// TwinCAT 3 PLC project WP_Controller
// ProgramVersion: 3.1.4024.0
// libraries:
//   CmpBitmapPool, * (System)
//   Tc2_EtherCAT, * (Beckhoff Automation GmbH)
//   Tc2_MC2, * (Beckhoff Automation GmbH)
//   Tc2_ModbusRTU, * (Beckhoff Automation GmbH)
//   Tc2_Standard, * (Beckhoff Automation GmbH)
//   Tc2_System, * (Beckhoff Automation GmbH)
//   Tc2_Utilities, * (Beckhoff Automation GmbH)
//   Tc3_Module, * (Beckhoff Automation GmbH)
//   Tc3_Vision, * (Beckhoff Automation GmbH)
// project tree:
//   DUTs/EtherCATDiagnostic/ E_EcDiacStatus.TcDUT (not stored), E_EcGetSlaveName.TcDUT (not stored), E_EcSystemStatus.TcDUT (not stored), ST_EcTerminalDiagInfo.TcDUT (not stored)
//   DUTs/TwinSAFE/ ST_AdsAddr.TcDUT (not stored)
//   DUTs/TwinSAFE/TwinSAFE_Connection/AX5805/ E_TsDiagnosisObjektsFA10AX5805.TcDUT, E_TsErrIndicesFA82AX5805.TcDUT, ST_TsConnectionInfoAX5805.TcDUT, ST_TsControlWordAX5805.TcDUT, ST_TsDiagObjectsFA10AX5805.TcDUT, ST_TsErrIndicesFA82AX5805.TcDUT, ST_TsSlaveInfoAX5805.TcDUT, ST_TsStatusWordAX5805.TcDUT
//   DUTs/TwinSAFE/TwinSAFE_Connection/EK1914/ ST_TsConnectionInfoEK1914.TcDUT, ST_TsDiagObjectsBitsEK1914.TcDUT, ST_TsDiagObjectsEK1914.TcDUT, ST_TsSlaveInfoEK1914.TcDUT
//   DUTs/TwinSAFE/TwinSAFE_Connection/EK1960/ ST_TsConnectionInfoEK1960.TcDUT, ST_TsDeviceInfoDataEK1960.TcDUT, ST_TsDiagObjectsEK1960.TcDUT, ST_TsSlaveInfoEK1960.TcDUT
//   DUTs/TwinSAFE/TwinSAFE_Connection/EL1904/ ST_TsConnectionInfoEL1904.TcDUT (not stored), ST_TsDiagObjectsBitsEL1904.TcDUT (not stored), ST_TsDiagObjectsEL1904.TcDUT (not stored), ST_TsSlaveInfoEL1904.TcDUT (not stored)
//   DUTs/TwinSAFE/TwinSAFE_Connection/EL1918/ ST_TsConnectionInfoEL1918.TcDUT, ST_TsDeviceInfoDataEL1918.TcDUT, ST_TsDiagObjectsEL1918.TcDUT, ST_TsSlaveInfoEL1918.TcDUT
//   DUTs/TwinSAFE/TwinSAFE_Connection/EL2904/ ST_TsConnectionInfoEL2904.TcDUT (not stored), ST_TsDiagObjectsBitsEL2904.TcDUT (not stored), ST_TsDiagObjectsEL2904.TcDUT (not stored), ST_TsSlaveInfoEL2904.TcDUT (not stored)
//   DUTs/TwinSAFE/TwinSAFE_Connection/EL2911/ ST_TsConnectionInfoEL2911.TcDUT, ST_TsDeviceInfoDataEL2911.TcDUT, ST_TsDiagObjectsEL2911.TcDUT, ST_TsSlaveInfoEL2911.TcDUT
//   DUTs/TwinSAFE/TwinSAFE_Connection/EL2912/ ST_TsConnectionInfoEL2912.TcDUT, ST_TsDeviceInfoDataEL2912.TcDUT, ST_TsDiagObjectsEL2912.TcDUT, ST_TsSlaveInfoEL2912.TcDUT
//   DUTs/TwinSAFE/TwinSAFE_Connection/EL3214/ ST_TsConnectionInfoEL3214.TcDUT, ST_TsSlaveInfoEL3214.TcDUT
//   DUTs/TwinSAFE/TwinSAFE_Connection/EL5021/ ST_TsConnectionInfoEL5021.TcDUT, ST_TsSlaveInfoEL5021.TcDUT
//   DUTs/TwinSAFE/TwinSAFE_Connection/EL6900/ ST_TsHardwareDiagC.TcDUT, ST_TsSlaveInfoEL6900.TcDUT
//   DUTs/TwinSAFE/TwinSAFE_Connection/EL6910/ ST_TsDeviceInfoDataC.TcDUT (not stored), ST_TsSlaveInfoEL6910.TcDUT (not stored)
//   DUTs/TwinSAFE/TwinSAFE_Connection/EP1957/ ST_TsConnectionInfoEP1957.TcDUT, ST_TsDeviceInfoDataEP1957.TcDUT, ST_TsDiagObjectsEP1957.TcDUT, ST_TsSlaveInfoEP1957.TcDUT
//   DUTs/TwinSAFE/TwinSAFE_Connection/ E_TsCycleDiagObj.TcDUT (not stored), ST_TsConnectionInfo12Byte.TcDUT (not stored), ST_TsConnectionInfo1Byte.TcDUT (not stored), ST_TsConnectionInfo2Byte.TcDUT (not stored), ST_TsConnectionInfo4Byte.TcDUT (not stored), ST_TsConnectionInfo8Byte.TcDUT (not stored), ST_TsSlave2Temp.TcDUT (not stored), ST_TsSlave3Temp.TcDUT (not stored), ST_TsSlaveAddress.TcDUT (not stored), ST_TsSlaveAddressCRC.TcDUT (not stored)
//   DUTs/TwinSAFE/TwinSAFE_Functionblocks/ E_TsFbType.TcDUT (not stored), ST_TsFbInfo.TcDUT (not stored)
//   DUTs/TwinSAFE/TwinSAFE_Group/ ST_TsGroupInfo.TcDUT (not stored)
//   GVLs/ GVL.TcGVL, IO.TcGVL
//   / PlcTask.TcTTO (not stored), VisionTask.TcTTO (not stored)
//   POUs/ FB_ClockPulse.TcPOU, FB_EnableAxes.TcPOU (not stored), FB_StrASCConversion.TcPOU (not stored), F_Scale.TcPOU (not stored), MAIN.TcPOU, PRG_LoadcellScaling.TcPOU, PRG_MotorDrive.TcPOU, PRG_PLCModbusRTU.TcPOU, PRG_PneumaticValves.TcPOU, PRG_PowerMeasurement.TcPOU, PRG_SafetyLightCurtain.TcPOU, PRG_Thermocouple.TcPOU, PRG_VfdModbusRtu.TcPOU, VISION.TcPOU, Vision_test.TcPOU
//   POUs/TwinSAFE/ FB_EcGetSlaveName.TcPOU, FB_TwinSafeConnectionEL1904.TcPOU (not stored), FB_TwinSafeConnectionEL2912.TcPOU, FB_TwinSafeConnectionEL6910.TcPOU (not stored), FB_TwinSafeFB.TcPOU (not stored), FB_TwinSafeGroup.TcPOU (not stored), FB_TwinSafeGroupExt.TcPOU (not stored)
// real-time tasks:
//   TASK PlcTask: cycle T#10ms, priority 20, ADS port 350
//   TASK VisionTask: cycle T#10ms, priority 21, ADS port 351
//   TASK VnTask ImgAcq (Camera1): cycle T#1ms, priority 5, ADS port 352
//   TASK VnTask ADS (Camera1): cycle T#10ms, priority 6, ADS port 353
//   TASK VnTask ImgAcq (FileSource1): cycle T#10ms, priority 7, ADS port 354
// motion (NC):
//   TASK NC-Task 1 SAF: cycle T#2ms, priority 4, ADS port 501
//   TASK NC-Task 1 SVB: cycle T#10ms, priority 8, ADS port 511
//   AXIS Axis 1 (id 1)
//     General: UnitName=°
//     Dynamic: AccelerationMaximum=52000, DecelerationMaximum=52000, Acceleration=49770, Deceleration=49770, Jerk=149310
//     Velo: RefSearch=331.8, RefSync=331.8, SlowManual=1659, FastManual=9954, Fast=33180, Maximum=33180
//     OtherSettings: AllowMotionCmdToSlave=true
//     encoder EncType=19
//       EncPara: ScaleFactorNumerator=360, ScaleFactorDenominator=1048576, MaxCount=#xffffffff
//         TimeComp: TimeCompMode=1, EncDelayCycles=4
//     drive DrvType=16
//       DrvPara: MaxCount=#xffffffff, DriveControlDWord=#x00020000
//         Analog: VeloReferenz=36498, VeloScale=32, TorqueSetpointScale=10, ScaleFactorActTorque=0.1
//         TimeComp: TaskDelayCycles=1
//     controller CtrType=1
//       CtrPara: PriorControlFactor=1
//         PosDiffControl: Enable=false
//         Observer: BandWidth=20
// I/O:
//   DEVICE Device 5 (EtherCAT), AmsNetId 169.254.69.6.6.1
//     Term 12 (EK1100) [EK1100 EtherCAT Coupler (2A E-Bus)]
//       Term 13 (EL1809) [EL1809 16Ch. Dig. Input 24V, 3ms]
//       Term 14 (EL2809-0015) [EL2809-0015 16Ch. Dig. Output 24V DC, 0.35A, not short-circuit proof]
//       Term 15 (EL6910) [EL6910, TwinSAFE PLC]
//       Term 16 (EL1904) [EL1904, 4 Ch. Safety Input 24V, TwinSAFE]
//         modules: Module 1 (FSOES)
//       Term 17 (EL2912) [EL2912, 2Ch. Safety Output 24V, 2A, TwinSAFE]
//         modules: Module 1 (FSOE), Module 2 (FSOUT), Module 3 (DEVICEIO), Module 4 (FSLOGIC)
//       Term 18 (EL3443) [EL3443 3Ch. Power Measuring]
//       Term 19 (EL3312) [EL3312 2Ch. Ana. Input Thermocouple (TC)]
//       Term 20 (EL6021) [EL6021 Interface (RS422/485)]
//       Term 21 (EL6021) [EL6021 Interface (RS422/485)]
//       Term 22 (EL9410) [EL9410 E-Bus Power Supplier  (Diagnostics)]
//       Term 23 (EL7221-9014) [EL7221-9014 1Ch. MDP742 Servo motor output stage with OCT (50V, 8A RMS) and STO input]
//       Term 24 (EL7221-9014) [EL7221-9014 1Ch. MDP742 Servo motor output stage with OCT (50V, 8A RMS) and STO input]
//       Term 25 (EL9512) [EL9512 Power supply terminal 12V]
//       Term 26 (EL3356-0010) [EL3356-0010 1Ch. Ana. Input Resistor Bridge Terminal, 24bit, High Precision]
//       Term 27 (EL9011) [EL9011 End Terminal]
// variable links:
//   NC-Task 1 SAF/Axes/Axis 1 <-> Device 5 (EtherCAT)/Term 12 (EK1100)/Term 23 (EL7221-9014)
//     Drive/Inputs/In/nDcOutputTime <-> InfoData/DcOutputShift
//     Drive/Inputs/In/nState1 <-> DRV Statusword/Statusword
//     Drive/Inputs/In/nState2 <-> DRV Statusword/Statusword @bit 8
//     Drive/Inputs/In/nState4 @bit 1 <-> WcState/InputToggle
//     Drive/Inputs/In/nState4 <-> WcState/WcState
//     Drive/Outputs/Out/nCtrl1 <-> DRV Controlword/Controlword
//     Drive/Outputs/Out/nCtrl2 <-> DRV Controlword/Controlword @bit 8
//     Drive/Outputs/Out/nDataOut2 <-> DRV Target velocity/Target velocity
//     Enc/Inputs/In/nDataIn1 <-> FB Position/Position
//     Enc/Inputs/In/nDcInputTime <-> InfoData/DcInputShift
//     Enc/Inputs/In/nState4 @bit 1 <-> WcState/InputToggle
//     Enc/Inputs/In/nState4 <-> WcState/WcState
//   WP_Controller/WP_Controller Instance <-> Device 5 (EtherCAT)/Term 12 (EK1100)/Term 14 (EL2809-0015)
//     PlcTask Outputs/GVL.bFan <-> Channel 9/Output
//     PlcTask Outputs/GVL.bLight <-> Channel 8/Output
//   WP_Controller/WP_Controller Instance <-> Device 5 (EtherCAT)/Term 12 (EK1100)/Term 18 (EL3443)
//     PlcTask Inputs/GVL.fActivePower <-> L1 Power/Active Power
//     PlcTask Inputs/GVL.fIL1 <-> L1 Basic/Current
//     VisionTask Inputs/GVL.fFrequency <-> Total Basic/Frequency
//     VisionTask Inputs/GVL.fUL1 <-> L1 Basic/Voltage
//     VisionTask Inputs/GVL.fcosphi1 <-> L1 Power/Power Factor
//   WP_Controller/WP_Controller Instance <-> Device 5 (EtherCAT)/Term 12 (EK1100)/Term 19 (EL3312)
//     PlcTask Inputs/GVL.nTemp <-> TC Inputs Channel 1/Value
//   WP_Controller/WP_Controller Instance <-> Device 5 (EtherCAT)/Term 12 (EK1100)/Term 20 (EL6021)
//     PlcTask Inputs/PRG_VfdModbusRtu.fbVfdMb.InData/D <-> COM TxPDO-Map Inputs/Data In 0
//     PlcTask Inputs/PRG_VfdModbusRtu.fbVfdMb.InData/D @bit {8..168 step 8} <-> COM TxPDO-Map Inputs/Data In {1..21}  (21 links)
//     PlcTask Inputs/PRG_VfdModbusRtu.fbVfdMb.InData/Status <-> COM TxPDO-Map Inputs/Status
//     PlcTask Outputs/PRG_VfdModbusRtu.fbVfdMb.OutData/Ctrl <-> COM RxPDO-Map Outputs/Ctrl
//     PlcTask Outputs/PRG_VfdModbusRtu.fbVfdMb.OutData/D <-> COM RxPDO-Map Outputs/Data Out 0
//     PlcTask Outputs/PRG_VfdModbusRtu.fbVfdMb.OutData/D @bit {8..168 step 8} <-> COM RxPDO-Map Outputs/Data Out {1..21}  (21 links)
//   WP_Controller/WP_Controller Instance <-> Device 5 (EtherCAT)/Term 12 (EK1100)/Term 21 (EL6021)
//     PlcTask Inputs/PRG_PLCModbusRTU.fbModbusMaster.InData/D <-> COM TxPDO-Map Inputs/Data In 0
//     PlcTask Inputs/PRG_PLCModbusRTU.fbModbusMaster.InData/D @bit {8..168 step 8} <-> COM TxPDO-Map Inputs/Data In {1..21}  (21 links)
//     PlcTask Inputs/PRG_PLCModbusRTU.fbModbusMaster.InData/Status <-> COM TxPDO-Map Inputs/Status
//     PlcTask Outputs/PRG_PLCModbusRTU.fbModbusMaster.OutData/Ctrl <-> COM RxPDO-Map Outputs/Ctrl
//     PlcTask Outputs/PRG_PLCModbusRTU.fbModbusMaster.OutData/D <-> COM RxPDO-Map Outputs/Data Out 0
//     PlcTask Outputs/PRG_PLCModbusRTU.fbModbusMaster.OutData/D @bit {8..168 step 8} <-> COM RxPDO-Map Outputs/Data Out {1..21}  (21 links)
//   WP_Controller/WP_Controller Instance <-> Device 5 (EtherCAT)/Term 12 (EK1100)/Term 26 (EL3356-0010)
//     PlcTask Inputs/GVL.uLoadCellRawValue <-> RMB Value (INT32)/Value
//   WP_Controller/WP_Controller Instance <-> NC-Task 1 SAF/Axes/Axis 1
//     PlcTask Inputs/GVL.stAxis1.NcToPlc <-> Outputs/ToPlc
//     PlcTask Outputs/GVL.stAxis1.PlcToNc <-> Inputs/FromPlc

// ---- DUTs/TwinSAFE/TwinSAFE_Connection/AX5805/E_TsDiagnosisObjektsFA10AX5805.TcDUT
TYPE E_TsDiagnosisObjektsFA10AX5805 :
(*******************************************************************************************************
Description			:	Reason for shutdown of CoE objects 0xFA10
Supported terminals : 	AX5805, AX5806
Documentation 		:	AX5805 / AX5806 TwinSAFE drive option cards for the AX5000 servo drive
Version/Date 		:	V1.6.1/15.03.2016
********************************************************************************************************)
(

	eFA10AX5805_NoErrorReaction					:= 16#0000,	(* Error reaction: no error reaction *)
	eFA10AX5805_ErrSafeTorqueOff				:= 16#0040,	(* Error reaction: STO (Safe Torque Off) *)
	eFA10AX5805_ErrSafeStop1					:= 16#0050,	(* Error reaction: SS1 (Safe Stop 1) *)

	eFA10AX5805_StatusWordIncorrect				:= 16#0100,	(* Shutdown reason: The status word was calculated incorrectly *)
	eFA10AX5805_ParametersWrongOrNotLoaded		:= 16#0200,	(* Shutdown reason: The parameters are wrong or not yet loaded *)
	eFA10AX5805_FSOEProtocolWrongState			:= 16#0300,	(* Shutdown reason: FSOE protocol not in state DATA *)
	eFA10AX5805_WrongDriveParameter				:= 16#0400,	(* Shutdown reason: Internal comparison failed. Please check the motor/drive dimensioning/parameterization *)
	eFA10AX5805_ExtCamDetectedUnexpectedly		:= 16#0500,	(* Reason for shutdown position detection: external cam detected unexpectedly *)
	eFA10AX5805_ExtCamRightSideCamWindow		:= 16#0600,	(* Reason for shutdown position detection: external cam detected to the right of the cam window *)
	eFA10AX5805_ExtCamLeftSideCamWindow			:= 16#0700,	(* Reason for shutdown position detection: external cam detected to the left of the cam window *)
	eFA10AX5805_MaxTraversingRangeExceeded		:= 16#0800,	(* Reason for shutdown position detection: the maximum traversing range was exceeded *)
	eFA10AX5805_SS1SwitchedOff					:= 16#5000,	(* Reason for shutdown safety function: The safety function SS1 has switched off *)
	eFA10AX5805_SOSSwitchedOff					:= 16#6800,	(* Reason for shutdown safety function: The safety function SOS has switched off *)
	eFA10AX5805_SSRSwitchedOff					:= 16#8000,	(* Reason for shutdown safety function: The safety function SSR has switched off *)
	eFA10AX5805_SLSSwitchedOff					:= 16#9000,	(* Reason for shutdown safety function: The safety function SLS has switched off *)
	eFA10AX5805_SLPSwitchedOff					:= 16#A000,	(* Reason for shutdown safety function: The safety function SLP has switched off *)
	eFA10AX5805_SMSSwitchedOff					:= 16#A800,	(* Reason for shutdown safety function: The safety function SMS has switched off *)
	eFA10AX5805_SLISwitchedOff					:= 16#B800,	(* Reason for shutdown safety function: The safety function SLI has switched off *)
	eFA10AX5805_SARSwitchedOff					:= 16#C000,	(* Reason for shutdown safety function: The safety function SAR has switched off *)
	eFA10AX5805_SMASwitchedOff					:= 16#C800,	(* Reason for shutdown safety function: The safety function SMA has switched off *)
	eFA10AX5805_SDIpSwitchedOff					:= 16#D000,	(* Reason for shutdown safety function: The safety function SDIp has switched off *)
	eFA10AX5805_SDInSwitchedOff					:= 16#D100	(* Reason for shutdown safety function: The safety function SDIn has switched off *)
	
);
END_TYPE
(* End *)

// ---- DUTs/TwinSAFE/TwinSAFE_Connection/AX5805/E_TsErrIndicesFA82AX5805.TcDUT
TYPE E_TsErrIndicesFA82AX5805 :
(*******************************************************************************************************
Description			:	Error indices in CoE objects 0xFA82
Supported terminals : 	AX5805, AX5806
Documentation 		:	AX5805 / AX5806 TwinSAFE drive option cards for the AX5000 servo drive
Version/Date 		:	V1.6.1/15.03.2016
********************************************************************************************************)
(

	eAX5805FA82_NoError									:=	16#0000,	

	eAX5805FA82_FAULT_MAXT_C1							:=	16#0001,	(* The temperature has exceeded the maximum permissible temperature (µC1) *)
	eAX5805FA82_FAULT_MAXT_C2							:=	16#0002,	(* The temperature has exceeded the maximum permissible temperature (µC2) *)
	eAX5805FA82_FAULT_MINT_C1							:=	16#0003,	(* The temperature has fallen below the minimum permissible temperature (µC1) *)
	eAX5805FA82_FAULT_MINT_C2							:=	16#0004,	(* The temperature has fallen below the minimum permissible temperature (µC2) *)

	eAX5805FA82_HW_ERR_MAX_VCC_C1						:=	16#0101,	(* The maximum supply voltage was exceeded (3.3 V) *)
	eAX5805FA82_HW_ERR_MAX_VCC_C2						:=	16#0102,	(* The maximum supply voltage was exceeded (3.3 V) *)
	eAX5805FA82_HW_ERR_MIN_VCC_C1						:=	16#0103,	(* The supply voltage fell below the minimum value (3.3 V) *)
	eAX5805FA82_HW_ERR_MIN_VCC_C2						:=	16#0104,	(* The supply voltage fell below the minimum value (3.3 V) *)

	eAX5805FA82_FAULT_MCTC1_TO							:=	16#0201,	(* The MCTests of µC1 were not carried out completely within the specified time *)
	eAX5805FA82_FAULT_MCTC2_TO							:=	16#0202,	(* The MCTests of µC2 were not carried out completely within the specified time *)
	eAX5805FA82_FAULT_TIMER_C1							:=	16#0203,	(* The global timer was not updated in time *)
	eAX5805FA82_FAULT_TIMER_C2							:=	16#0204,	(* The global timer was not updated in time *)
	eAX5805FA82_FAULT_TS_WDG_TO_C1						:=	16#020C,	(* The TwinSAFE module was not called within the watchdog time *)
	eAX5805FA82_FAULT_TS_WDG_TO_C2						:=	16#020D,	(* The TwinSAFE module was not called within the watchdog time *)
	eAX5805FA82_FAULT_RESET_MC1							:=	16#020E,	(* A reset has occurred in the operation of the controller for µC1. µC2 was not reset thereby *)
	
	eAX5805FA82_FAULT_SERCOMC2							:=	16#0300,	(* An error occurred in the SerComP24C2 module during data transmission *)

	eAX5805FA82_FAULT_SERCOM_1							:=	16#0401,	(* An error occurred in the SerComP24C1 module during data transmission *)
	eAX5805FA82_FAULT_SERCOM_2							:=	16#0402,	(* An error occurred in the SerComP24C1 module during data transmission *)
	eAX5805FA82_FAULT_SERCOM_3							:=	16#0403,	(* An error occurred in the SerComP24C1 module during data transmission *)
	eAX5805FA82_FAULT_SERCOM_4							:=	16#0404,	(* An error occurred in the SerComP24C1 module during data transmission *)
	eAX5805FA82_FAULT_SERCOM_5							:=	16#0405,	(* An error occurred in the SerComP24C1 module during data transmission *)
	eAX5805FA82_FAULT_SERCOM_6							:=	16#0406,	(* An error occurred in the SerComP24C1 module during data transmission *)
	eAX5805FA82_FAULT_SERCOM_7							:=	16#0407,	(* An error occurred in the SerComP24C1 module during data transmission *)
	eAX5805FA82_FAULT_SERCOM_8							:=	16#0408,	(* An error occurred in the SerComP24C1 module during data transmission *)
	eAX5805FA82_FAULT_SERCOM_9							:=	16#0409,	(* An error occurred in the SerComP24C1 module during data transmission *)
	eAX5805FA82_FAULT_SERCOM_A							:=	16#040A,	(* An error occurred in the SerComP24C1 module during data transmission *)
	eAX5805FA82_FAULT_SERCOM_B							:=	16#040B,	(* An error occurred in the SerComP24C1 module during data transmission *)

	eAX5805FA82_FAULT_TEMPSENSOR_1						:=	16#0501,	(* Error in the communication with one of the temperature sensors *)
	eAX5805FA82_FAULT_TEMPSENSOR_2						:=	16#0502,	(* Error in the communication with one of the temperature sensors *)
	eAX5805FA82_FAULT_TEMPSENSOR_3						:=	16#0503,	(* Error in the communication with one of the temperature sensors *)
	eAX5805FA82_FAULT_TEMPSENSOR_4						:=	16#0504,	(* Error in the communication with one of the temperature sensors *)
	eAX5805FA82_FAULT_TEMPSENSOR_5						:=	16#0505,	(* Error in the communication with one of the temperature sensors *)
	eAX5805FA82_FAULT_TEMPSENSOR_6						:=	16#0506,	(* Error in the communication with one of the temperature sensors *)
	eAX5805FA82_FAULT_TEMPSENSOR_7						:=	16#0507,	(* Error in the communication with one of the temperature sensors *)

	eAX5805FA82_FAULT_OUTPUTCOMPARE						:=	16#0601,	(* The values output by µC1 and µC2 differ *)
	eAX5805FA82_FAULT_OUTPUTCOMPAREC2					:=	16#0602,	(* The values output by µC1 and µC2 differ *)

	eAX5805FA82_HW_ERR_MIN_VCC_FPGA						:=	16#0700,	(* The FPGA supply voltage fell below the minimum value (5 V) *)
	eAX5805FA82_HW_ERR_MAX_VCC_FPGA						:=	16#0701,	(* The FPGA supply voltage exceeded the maximum value (5 V) *)

	eAX5805FA82_FAULT_FEEDBACK_C1						:=	16#0710,	(* An error was detected in the feedback channels of µC1 *)
	eAX5805FA82_FAULT_FEEDBACK_C2						:=	16#0711,	(* An error was detected in the feedback channels of µC2 *)

	eAX5805FA82_FAULT_Parameter_C1						:=	16#0720,	(* General parameter error µC1 *)
	eAX5805FA82_FAULT_Parameter_C2						:=	16#0721,	(* General parameter error µC2 *)
	eAX5805FA82_FAULT_Parameter_C1_DRIVE_PROFILE		:=	16#0722,	(* Parameter: unknown parameter index µC1 drive profile *)
	eAX5805FA82_FAULT_Parameter_C1_VENDOR_SPECIFIC		:=	16#0723,	(* Parameter: unknown parameter index µC1 vendor-specific *)
	eAX5805FA82_FAULT_Parameter_C2_DRIVE_PROFILE		:=	16#0724,	(* Parameter: unknown parameter index µC2 drive profile *)
	eAX5805FA82_FAULT_Parameter_C2_VENDOR_SPECIFIC		:=	16#0725,	(* Parameter: unknown parameter index µC2 vendor-specific *)
	eAX5805FA82_FAULT_PDO_MAPPING_FSOE_COMMAND			:=	16#0726,	(* PDO mapping axis 1/2: FSOE COMMAND error *)
	eAX5805FA82_FAULT_PDO_MAPPING_LENGTH				:=	16#0727,	(* PDO mapping axis 1: Length_Error *)
	eAX5805FA82_FAULT_PDO_MAPPING_STO_K1				:=	16#0728,	(* PDO mapping axis 1: STO error *)
	eAX5805FA82_FAULT_PDO_MAPPING_SS1_1_K1				:=	16#0729,	(* PDO mapping axis 1: Error SS1_1 *)
	eAX5805FA82_FAULT_PDO_MAPPING_SS2_1_K1				:=	16#072A,	(* PDO mapping axis 1: Error SS2_1 *)
	eAX5805FA82_FAULT_PDO_MAPPING_SOS_1_K1				:=	16#072B,	(* PDO mapping axis 1: SS2_1 error *)
	eAX5805FA82_FAULT_PDO_MAPPING_SSR_1_K1				:=	16#072C,	(* PDO mapping axis 1: SSR_1 error *)
	eAX5805FA82_FAULT_PDO_MAPPING_SDIp_K1				:=	16#072D,	(* PDO mapping axis 1: SDIp error *)
	eAX5805FA82_FAULT_PDO_MAPPING_SDIn_K1				:=	16#072E,	(* PDO mapping axis 1: SDIn error *)
	eAX5805FA82_FAULT_PDO_MAPPING_Error_ACK_K1			:=	16#072F,	(* PDO mapping axis 1: Error_ACK error *)
	
	eAX5805FA82_FAULT_PDO_MAPPING_Error_CRC0			:=	16#0730,	(* PDO mapping axis 1/2: FSOE CRC0 error *)
	eAX5805FA82_FAULT_PDO_MAPPING_STO_K2				:=	16#0731,	(* PDO mapping axis 2: STO error *)
	eAX5805FA82_FAULT_PDO_MAPPING_SS1_1_K2				:=	16#0732,	(* PDO mapping axis 2: Error SS1_1 *)
	eAX5805FA82_FAULT_PDO_MAPPING_SS2_1_K2				:=	16#0733,	(* PDO mapping axis 2: Error SS2_1 *)
	eAX5805FA82_FAULT_PDO_MAPPING_SOS_1_K2				:=	16#0734,	(* PDO mapping axis 2: SS2_1 error *)
	eAX5805FA82_FAULT_PDO_MAPPING_SSR_1_K2				:=	16#0735,	(* PDO mapping axis 2: SSR_1 error *)
	eAX5805FA82_FAULT_PDO_MAPPING_SDIp_K2				:=	16#0736,	(* PDO mapping axis 2: SDIp error *)
	eAX5805FA82_FAULT_PDO_MAPPING_SDIn_K2				:=	16#0737,	(* PDO mapping axis 2: SDIn error *)
	eAX5805FA82_FAULT_PDO_MAPPING_Error_ACK_K2			:=	16#0738,	(* PDO mapping axis 2: Error_ACK error *)
	eAX5805FA82_FAULT_PDO_MAPPING_Error_CRC1			:=	16#0739,	(* PDO mapping axis 2: FSOE CRC1 error *)
	eAX5805FA82_FAULT_PDO_MAPPING_Error_ConnID			:=	16#073A,	(* PDO mapping axis 1/2: FSOE ConnID error *)
	eAX5805FA82_FAULT_PDO_MAPPING_SSM_1_K1				:=	16#073B,	(* PDO mapping axis 1: SSM_1_K1 error *)
	eAX5805FA82_FAULT_PDO_MAPPING_SSM_1_K2				:=	16#073C,	(* PDO mapping axis 2: SSM_1_K2 error *)
	eAX5805FA82_FAULT_PDO_MAPPING_SSM_2_K1				:=	16#073D,	(* PDO mapping axis 1: SSM_2_K1 error *)
	eAX5805FA82_FAULT_PDO_MAPPING_SSM_2_K2				:=	16#073E,	(* PDO mapping axis 2: SSM_2_K2 error *)	

	eAX5805FA82_FAULT_WRONG_MOTORCONSTRUCTIONTYPE_K1	:=	16#0740,	(* Register communication: parameterized motor type for axis 1 does not correspond to the connected motor *)
	eAX5805FA82_FAULT_UNKNOWN_MOTOR_TYPE_K1				:=	16#0741,	(* Register communication: parameterized motor type for axis 1 is unknown *)
	eAX5805FA82_FAULT_WRONG_MOTORCONSTRUCTIONTYPE_K2	:=	16#0742,	(* Register communication: parameterized motor type for axis 2 does not correspond to the connected motor *)
	eAX5805FA82_FAULT_UNKNOWN_MOTOR_TYPE_K2				:=	16#0743,	(* Register communication: parameterized motor type for axis 2 is unknown *)
	eAX5805FA82_FAULT_NUM_OF_POLEPAIRS_K1				:=	16#0744,	(* Register communication: parameterized number of pole pairs for axis 1 does not correspond to the connected motor *)
	eAX5805FA82_FAULT_NUM_OF_POLEPAIRS_K2				:=	16#0745,	(* Register communication: parameterized number of pole pairs for axis 2 does not correspond to the connected motor *)
	eAX5805FA82_FAULT_WRONG_MOTOR_CONFIGURED_K1			:=	16#0746,	(* Register communication: parameterized motor type for axis 1 does not correspond to the connected motor *)
	eAX5805FA82_FAULT_WRONG_MOTOR_CONFIGURED_K2			:=	16#0747,	(* Register communication: parameterized motor type for axis 2 does not correspond to the connected motor *)
	eAX5805FA82_FAULT_RXPDO_LENGTH						:=	16#0748,	(* PDO mapping: RXPDO length is wrong *)
	eAX5805FA82_FAULT_TXPDO_LENGTH						:=	16#0749,	(* PDO mapping: TXPDO length is wrong *)
	eAX5805FA82_FAULT_UNKNOWN_RXPDO_INDEX				:=	16#074A,	(* PDO mapping: RXPDO index is unknown *)
	eAX5805FA82_FAULT_UNKNOWN_TXPDO_INDEX				:=	16#074B,	(* PDO mapping: TXPDO index is unknown *)
	eAX5805FA82_FAULT_WRONG_NUMBER_OF_AXLE				:=	16#074C, 	(* The parameterized number of axes does not correspond to the number detected *)

	eAX5805FA82_FAULT_CRC_INIT_C1						:=	16#1001,	(* An incorrect checksum at µC1 was determined during PowerOn reset *)
	eAX5805FA82_FAULT_CRC_INIT_C2						:=	16#1002,	(* An incorrect checksum at µC2 was determined during PowerOn reset *)
	eAX5805FA82_FAULT_CRC_C1							:=	16#1003,	(* An incorrect checksum was determined for µC1 during operation *)
	eAX5805FA82_FAULT_CRC_C2							:=	16#1004,	(* An incorrect checksum was determined for µC2 during operation *)
	eAX5805FA82_FAULT_RAM_C1							:=	16#1011,	(* An error occurred during the RAM test of µC1 - Typical error reaction time (125µs) *)
	eAX5805FA82_FAULT_RAM_C2							:=	16#1012,	(* An error occurred during the RAM test of µC2 - Typical error reaction time (125µs) *)
	eAX5805FA82_FAULT_RAM_CHECKERBOARD_C1				:=	16#1013,	(* An error occurred during the RAM test of µC1 *)
	eAX5805FA82_FAULT_RAM_CHECKERBOARD_C2				:=	16#1014,	(* An error occurred during the RAM test of µC2 *)
	eAX5805FA82_FAULT_GLBL_TMR							:=	16#1021,	(* The global timer is not working correctly - Typical error reaction time (125µs) *)
	eAX5805FA82_FAULT_SPLIM1							:=	16#1031,	(* Stack overruns are no longer being intercepted correctly *)
	eAX5805FA82_FAULT_SPLIM2							:=	16#1032,	(* Stack overruns are no longer being intercepted correctly *)

	eAX5805FA82_FAULT_OPCT_GRP_C1						:=	16#1100,	(* The opcode test for µC1 has failed *)

	eAX5805FA82_FAULT_OPCT_GRP_C2						:=	16#1300,	(* The opcode test for µC2 has failed *)

	eAX5805FA82_FAULT_ESS_CRC_C1						:=	16#1801,	(* Different check sums were determined in the TwinSAFE telegrams *)
	eAX5805FA82_FAULT_ESS_CRC_C2						:=	16#1802,	(* Different check sums were determined in the TwinSAFE telegrams *)
	eAX5805FA82_FAULT_SW_MAIN1_C1						:=	16#1803,	(* The default case of the main loop of µC1 was called *)
	eAX5805FA82_FAULT_SW_MAIN1_C2						:=	16#1804,	(* The default case of the main loop of µC2 was called *)
	eAX5805FA82_FAULT_ESLCONID_PRJCRCRD					:=	16#1805,	(* The Connection ID is not zero when reading the project CRC *)
	eAX5805FA82_FAULT_ESLCONID_PRJCRCWR					:=	16#1806,	(* The Connection ID is not zero when writing the project CRC *)
	eAX5805FA82_FAULT_SIZE_EEVONDOR_EXID				:=	16#1807,	(* An address was accessed that lies outside the vendor range in the EEPROM *)

	eAX5805FA82_FAULT_COM_C1C2							:=	16#5100,	(* Communication between µC1 and µC2 is disturbed *)
	eAX5805FA82_FAULT_ISR_SNT_FEEDBACK					:=	16#5101,	(* High priority ISR: communication interrupted: switched mode power supply feedback - Typical error reaction time (125µs) *)
	eAX5805FA82_FAULT_ISR_ANGLE_K1						:=	16#5102,	(* High priority ISR: communication interrupted: axis 1 angle - Typical error reaction time (125µs) *)
	eAX5805FA82_FAULT_ISR_ANGLE_K2						:=	16#5103,	(* High priority ISR: communication interrupted: axis 2 angle - Typical error reaction time (125µs) *)
	eAX5805FA82_FAULT_ISR_DELTA_K1						:=	16#5104,	(* High priority ISR: communication interrupted: axis 1 distance travelled - Typical error reaction time (125µs) *)
	eAX5805FA82_FAULT_ISR_DELTA_K2						:=	16#5105,	(* High priority ISR: communication interrupted: axis 2 distance travelled - Typical error reaction time (125µs) *)
	eAX5805FA82_FAULT_ISR_VELO_K1						:=	16#5106,	(* High priority ISR: communication interrupted: axis 1 velocity - Typical error reaction time (125µs) *)
	eAX5805FA82_FAULT_ISR_VELO_K2						:=	16#5107,	(* High priority ISR: communication interrupted: axis 2 velocity - Typical error reaction time (125µs) *)
	eAX5805FA82_FAULT_ISR_TEST_FEEDBACK					:=	16#5108,	(* High priority ISR: communication interrupted: feedback from switch-off channels - Typical error reaction time (125µs) *)
	eAX5805FA82_FAULT_TIMEOUT_REG_AX5000_CONTROL		:=	16#5109,	(* Register communication: AX5000 does not answer in time: Controlword *)
	eAX5805FA82_FAULT_TIMEOUT_REG_AX5000_STATUS			:=	16#510A,	(* Register communication: AX5000 does not answer in time: Statusword *)
	eAX5805FA82_FAULT_TIMEOUT_REG_AX5000_REGADR			:=	16#510B,	(* Register communication: AX5000 does not answer in time: Register address *)
	eAX5805FA82_FAULT_TIMEOUT_REG_AX5000_REGDATA		:=	16#510C,	(* Register communication: AX5000 does not answer in time: Register data *)
	eAX5805FA82_FAULT_TIMEOUT_REG_AX5000_CRC			:=	16#510D,	(* Register communication: AX5000 does not answer in time: CRC *)
	eAX5805FA82_FAULT_UNKNOWN_AX5000_INTERFACE			:=	16#510E,	(* Register communication: unknown interface to the AX5000 *)
	eAX5805FA82_FAULT_COMERROR_AX5000_INTERFACE			:=	16#510F,	(* Register communication: the interface to the AX5000 has a communication error *)
	eAX5805FA82_FAULT_WRITE_HW_VERSION_AX5805_0			:=	16#5110,	(* Values could not be written to the register in the AX5000 *)
	eAX5805FA82_FAULT_WRITE_HW_VERSION_AX5805_1			:=	16#5111,	(* Values could not be written to the register in the AX5000 *)
	eAX5805FA82_FAULT_WRITE_HW_VERSION_AX5805_2			:=	16#5112,	(* Values could not be written to the register in the AX5000 *)
	eAX5805FA82_FAULT_WRITE_HW_VERSION_AX5805_3			:=	16#5113,	(* Values could not be written to the register in the AX5000 *)
	eAX5805FA82_FAULT_EXT_ADC_ADDRESS					:=	16#5114,	(* High priority ISR: External ADC: an impermissible address was read *)
	eAX5805FA82_FAULT_REGISTER_AX5000_CRC_ERROR			:=	16#5115,	(* Register communication with the AX5000: telegram has a CRC error *)
	eAX5805FA82_FAULT_CYCLIC_AX5000_CRC_ERROR			:=	16#5116,	(* High priority ISR: cyclic communication with the AX5000: telegram has a CRC error - Typical error reaction time (125µs) *)
	eAX5805FA82_FAULT_UNKNOWN_REGISTER_ADDRESS			:=	16#5117,	(* Register communication: Addressed register is unknown *)
	eAX5805FA82_FAULT_AX5000_NOT_READY					:=	16#5118,	(* High priority ISR: cyclic communication with the AX5000: AX5000 signals a communication error - Typical error reaction time (125µs) *)
	eAX5805FA82_FAULT_C1C2_SYNC_LOST					:=	16#5119,	(* High priority ISR: cyclic communication between µC1 and µC2: Communication error - Typical error reaction time (125µs) *)

	eAX5805FA82_FAULT_SET_MAPPED_STATE					:=	16#5C00,	(* Mapped safety functions: error while setting the state *)
	eAX5805FA82_FAULT_RESET_MAPPED_STATE				:=	16#5C01,	(* Mapped safety functions: error while resetting the state *)
	eAX5805FA82_FAULT_MAPPED_FUNCTION					:=	16#5C02,	(* Mapped safety functions: invalid mapping, function does not exist *)
	eAX5805FA82_FAULT_MAPPED_INSTANCE					:=	16#5C03,	(* Mapped safety functions: invalid mapping, instance does not exist *)

	eAX5805FA82_FAULT_STO_MODE							:=	16#5E02,	(* The requested STO mode is invalid *)
	eAX5805FA82_FAULT_SDI_MODE							:=	16#5E03,	(* The requested SDI mode is invalid *)
	eAX5805FA82_FAULT_UNDEFINED_ERRORREACTION			:=	16#5E04,	(* Error reaction: invalid error reaction, error reaction does not exist *)

	eAX5805FA82_FAULT_CRC_COMPARE_C1					:=	16#5F00,	(* Incorrect checksum detected during comparison by µC1 *)
	eAX5805FA82_FAULT_CRC_COMPARE_C2					:=	16#5F01,	(* Incorrect checksum detected during comparison by µC2 *)
	eAX5805FA82_FAULT_TMR2_INTERRUPT_C1					:=	16#5F02,	(* MC_Test: Timer2 has triggered an interrupt on µC1. HighPrioISR was not called in time *)
	eAX5805FA82_FAULT_TMR2_INTERRUPT_C2					:=	16#5F03,	(* MC_Test: Timer2 has triggered an interrupt on µC2. HighPrioISR was not called in time *)
	eAX5805FA82_FAULT_SWITCHOFF_TEST					:=	16#5F04,	(* MC_Test: the test of the switch-off channels has failed *)
	eAX5805FA82_FAULT_NO_SYNC							:=	16#5F05,	(* No SYNC signal *)
	eAX5805FA82_FAULT_UNKNOWN_AXLE						:=	16#5F06,	(* The requested axis is unknown *)
	eAX5805FA82_FAULT_FPGA_C2							:=	16#5F07,	(* The status of the FPGA is incorrect *)
	eAX5805FA82_FAULT_ANGLE_FORMAT_C1					:=	16#5F08,	(* The angles OF µC1 read-in have the wrong format - Typical error reaction TIME (125µS) *)
	eAX5805FA82_FAULT_ANGLE_FORMAT_C2					:=	16#5F09,	(* The angles of µC2 read-in have the wrong format - Typical error reaction time (125µs) *)
	eAX5805FA82_FAULT_SAFE_MAIN_STATE					:=	16#5F0A,	(* Unknown state requested *)
	eAX5805FA82_FAULT_STARTUP_FAILED					:=	16#5F0B,	(* Error during start-up *)
	eAX5805FA82_FAULT_MOTION_DETECTION					:=	16#5F0C,	(* Motion detection error - Typical error reaction time (125µs) *)

	eAX5805FA82_FAULT_PARAMETER_FSOE_VENDOR_ID			:=	16#6000,	(* Incorrect vendor ID transmitted *)
	eAX5805FA82_FAULT_PARAMETER_FSOE_MODULE_IDENT		:=	16#6001,	(* Incorrect module ID transmitted *)
	eAX5805FA82_FAULT_PARAMETER_FSOE_CRC				:=	16#6002		(* CRC of the AX5805 parameters does not match the transmitted CRC (please check parameters; if necessary, activate System Manager configuration and reload safety project into the EL69xx) *)
);
END_TYPE
(* End *)

// ---- DUTs/TwinSAFE/TwinSAFE_Connection/AX5805/ST_TsConnectionInfoAX5805.TcDUT
TYPE ST_TsConnectionInfoAX5805 :
(*******************************************************************************************************
Description			:	Connection information data of EtherCAT Slaves with 4 byte input and 4 byte output safe data  
Supported terminals : 	AX5805(2 Axis)
Date 				:	04.11.2018
********************************************************************************************************)
STRUCT

	nState  								:USINT;
	nDiag 	 								:USINT;
	nInOutSafeDataByte1						:BYTE;
	nInOutSafeDataByte2						:BYTE;
	nInOutSafeDataByte3						:BYTE;
	nInOutSafeDataByte4						:BYTE;
	nInOutSafeDataByte5 					:BYTE;
	nInOutSafeDataByte6 					:BYTE;
	nInOutSafeDataByte7 					:BYTE;
	nInOutSafeDataByte8 					:BYTE;

END_STRUCT
END_TYPE
(* End *)

// ---- DUTs/TwinSAFE/TwinSAFE_Connection/AX5805/ST_TsControlWordAX5805.TcDUT
TYPE ST_TsControlWordAX5805 :
(*******************************************************************************************************
Description			:	Standard control Word of AX5805/6 terminal
Supported terminals : 	AX5805, AX5806
Documentation 		:	AX5805 / AX5806 TwinSAFE drive option cards for the AX5000 servo drive
Version/Date 		:	V1.6.1/15.03.2016
********************************************************************************************************)
STRUCT
	
	bSafeTorqueOff_STO 						:BOOL;
	bSafeStop1_SS1_1 						:BOOL;
	bSafeStop2_SS2_1 						:BOOL;
	bSafeOperatingStop_SOS_1 				:BOOL;
	bSafeSpeedRange_SSR_1 					:BOOL;
	bSafeDirectionPositive_SDIp				:BOOL;
	bSafeDirectionNegative_SDIn				:BOOL;
	bErrorAcknowledge_ErrAck				:BOOL;
	bNotInUseBit8	 						:BOOL;
	bNotInUseBit9	 						:BOOL;
	bNotInUseBit10	 						:BOOL;
	bNotInUseBit11	 						:BOOL;
	bNotInUseBit12	 						:BOOL;
	bNotInUseBit13	 						:BOOL;
	bNotInUseBit14	 						:BOOL;
	bNotInUseBit15				 			:BOOL;
	
END_STRUCT
END_TYPE
(* End *)

// ---- DUTs/TwinSAFE/TwinSAFE_Connection/AX5805/ST_TsDiagObjectsFA10AX5805.TcDUT
TYPE ST_TsDiagObjectsFA10AX5805 :
(*******************************************************************************************************
Description			:	Reason for shutdown of CoE objects 0xFA10
Supported terminals : 	AX5805, AX5806
Documentation 		:	AX5805 / AX5806 TwinSAFE drive option cards for the AX5000 servo drive
Version/Date 		:	V1.6.1/15.03.2016
********************************************************************************************************)
STRUCT

	nDummyData1								:ARRAY[0..3] OF UINT;
	nSoftwareCrcC1							:UINT;
	nSoftwareCrcC2							:UINT;
	nReasonForShutdownAxis1					:UINT;
	nReasonForShutdownAxis2					:UINT;
	
END_STRUCT
END_TYPE
(* End *)

// ---- DUTs/TwinSAFE/TwinSAFE_Connection/AX5805/ST_TsErrIndicesFA82AX5805.TcDUT
TYPE ST_TsErrIndicesFA82AX5805 :
(*******************************************************************************************************
Description			:	Error indices in CoE objects 0xFA82
Supported terminals : 	AX5805, AX5806
Documentation 		:	AX5805 / AX5806 TwinSAFE drive option cards for the AX5000 servo drive
Version/Date 		:	V1.6.1/15.03.2016
********************************************************************************************************)
STRUCT

(* Diagnosis motion contoler 1/2 *)
	nDiagnosisMC1							:UINT;
	nDiagnosisMC2							:UINT;

(* Error motion contoler 1/2 *)
	nErrorMC1								:UINT;
	nErrorMC2								:UINT;

END_STRUCT
END_TYPE
(* End *)

// ---- DUTs/TwinSAFE/TwinSAFE_Connection/AX5805/ST_TsSlaveInfoAX5805.TcDUT
TYPE ST_TsSlaveInfoAX5805 :
STRUCT
	
(* act_EcSlaveIdentify *)
	sEcSlaveType							:STRING(15);
	sEcSlaveName							:STRING(31) := '';
	bSlaveIdentify							:BOOL;
	bSlaveTypeError							:BOOL;
	
(* act_ConnectionState *)
	sState									:STRING;
	
(* act_ConnectionDiag *)
	sDiag									:STRING;
	sFault									:STRING;						(* FailSafe Error (Hardware)*)
	bError									:BOOL;							(* TwinSAFE-Error *)
	
(* act_ReadDiagObjects *)
	stSlaveTemp								:ST_TsSlave2Temp;
	bTempWarning							:BOOL;							(* Temperature warning: T1, T2 *)

	eErrIndicesFA82ErrorMC1					:E_TsErrIndicesFA82AX5805;
	eErrIndicesFA82ErrorMC2					:E_TsErrIndicesFA82AX5805;
	eErrIndicesFA82DiagnosisMC1				:E_TsErrIndicesFA82AX5805;
	bErrIndicesFA82DiagnosisMC1Err			:BOOL;
	eErrIndicesFA82DiagnosisMC2				:E_TsErrIndicesFA82AX5805;
	bErrIndicesFA82DiagnosisMC2Err			:BOOL;	

	eDiagObjFA10LowByteMC1					:E_TsDiagnosisObjektsFA10AX5805;
	eDiagObjFA10HighByteMC1					:E_TsDiagnosisObjektsFA10AX5805;
	eDiagObjFA10LowByteMC2					:E_TsDiagnosisObjektsFA10AX5805;
	eDiagObjFA10HighByteMC2					:E_TsDiagnosisObjektsFA10AX5805;
	
(* act_Signals *)
	stSignalStatusMC1						:ST_TsStatusWordAX5805;
	stSignalControlStatusMC1				:ST_TsControlWordAX5805;
	stSignalStatusMC2						:ST_TsStatusWordAX5805;
	stSignalControlStatusMC2				:ST_TsControlWordAX5805;

END_STRUCT
END_TYPE

// ---- DUTs/TwinSAFE/TwinSAFE_Connection/AX5805/ST_TsStatusWordAX5805.TcDUT
TYPE ST_TsStatusWordAX5805 :
(*******************************************************************************************************
Description			:	Standard status Word of AX5805/6 terminal
Supported terminals : 	AX5805, AX5806
Documentation 		:	AX5805 / AX5806 TwinSAFE drive option cards for the AX5000 servo drive
Version/Date 		:	V1.6.1/15.03.2016
********************************************************************************************************)
STRUCT
	
	bSafeTorqueOff_STO 						:BOOL;
	bSafeSpeedMonitor_SSM_1					:BOOL;
	bSafeSpeedMonitor_SSM_2					:BOOL;
	bSafeOperatingStop_SOS_1 				:BOOL;
	bSafeSpeedRange_SSR_1 					:BOOL;
	bSafeDirectionPositive_SDIp				:BOOL;
	bSafeDirectionNegative_SDIn				:BOOL;
	bErrorAcknowledge_ErrAck				:BOOL;
	bNotInUseBit8	 						:BOOL;
	bNotInUseBit9	 						:BOOL;
	bNotInUseBit10	 						:BOOL;
	bNotInUseBit11	 						:BOOL;
	bNotInUseBit12	 						:BOOL;
	bNotInUseBit13	 						:BOOL;
	bNotInUseBit14	 						:BOOL;
	bNotInUseBit15	 						:BOOL;

END_STRUCT
END_TYPE
(* End *)

// ---- DUTs/TwinSAFE/TwinSAFE_Connection/EK1914/ST_TsConnectionInfoEK1914.TcDUT
//{attribute 'pack_mode' := '0'}
TYPE ST_TsConnectionInfoEK1914 :
(*******************************************************************************************************
Description			:	Connection information data of EtherCAT Slaves with 2 byte input and 1 byte output safe data  
Supported terminals : 	EK1914
Date 				:	04.11.2018
********************************************************************************************************)
STRUCT

	nState  								:USINT;
	nDiag 	 								:USINT;
	nInOutSafeDataByte1						:BYTE;
	nInOutSafeDataByte2						:BYTE;

END_STRUCT
END_TYPE
(* End *)

// ---- DUTs/TwinSAFE/TwinSAFE_Connection/EK1914/ST_TsDiagObjectsBitsEK1914.TcDUT
TYPE ST_TsDiagObjectsBitsEK1914 :
(*******************************************************************************************************
Description			:	Index 16#800E Diagnostic objects
Supported terminals : 	EK1914
Documentation 		:	EK1914 TwinSAFE input/output terminal with 2 fail-safe inputs and 2 fail-safe outputs
Version/Date 		:	V1.2.0/08.03.2016
********************************************************************************************************)
STRUCT

(* Sensor test error *)
	bErrInput1								:BOOL;	(* Error input 1 - Bit0 - Error at input 1 *)
	bErrInput2								:BOOL;	(* Error input 2 - Bit1 - Error at input 2 *)

(* Error during two channel evaluation *)
	bErrFirstInputPair						:BOOL;	(* Error input 1..2 - Bit0 - Error in the first input pair *)

(* Error in the safety mat operating mode: input pair disagree *)
	bMatOpModeErrFirstInputPair				:BOOL;	(* Error input 1..2 - Bit1, Bit0 - Mat operating mode - Error in the first input pair *)

(* Error in the safety mat operating mode: external supply *)
	bMatOpModeExtSupplyErrInput1			:BOOL;	(* Error input 1 - Bit0 - Mat operating mode external supply - Error at input 1 *)
	bMatOpModeExtSupplyErrInput2			:BOOL;	(* Error input 2 - Bit1 - Mat operating mode external supply - Error at input 2 *)

(* Diagnosis μC1 *)
	bCcErrOutput1							:BOOL;	(* Diagnosis μC1 - Value  5    - Cross-circuit output 1 and output 2 *)
	bCcErrOutput2							:BOOL;	(* Diagnosis μC1 - Value  6    - Cross-circuit output 1 and output 2 *)
	bOvervoltage							:BOOL;	(* Diagnosis μC1 - Value 10    - Overvoltage *)
	bUndervoltage							:BOOL;	(* Diagnosis μC1 - Value 11    - Undervoltage *)
	bErrTestFieldVolSitches					:BOOL;	(* Diagnosis μC1 - Value 21-27 - Error when testing the field voltage switches *)
	bErrStartUpOutputCircuit				:BOOL;	(* Diagnosis μC1 - Value 30-33 - Start-up of the output circuit failed *)

	bExtSupply0VOutput1MicroC1				:BOOL;	(* Diagnosis μC1 - Value 101   - External supply 0 V output 1, detected with set output *)
	bExtSupply24VOutput1MicroC1				:BOOL;	(* Diagnosis μC1 - Value 102   - External supply 24 V output 1 *)
	bExtSupply0VOutput2MicroC1				:BOOL;	(* Diagnosis μC1 - Value 103   - External supply 0 V output 2, detected with set output *)
	bExtSupply24VOutput2MicroC1				:BOOL;	(* Diagnosis μC1 - Value 104   - External supply 24 V output 2 *)

(* Diagnosis μC2 *)
	bExtSupply0VOutput1MicroC2				:BOOL;	(* Diagnosis μC2 - Value 201 - External supply 0 V output 1, detected with set output *)
	bExtSupply24VOutput1MicroC2				:BOOL;	(* Diagnosis μC2 - Value 202 - External supply 24 V output 1 *)
	bExtSupply0VOutput2MicroC2				:BOOL;	(* Diagnosis μC2 - Value 203 - External supply 0 V output 2, detected with set output *)
	bExtSupply24VOutput2MicroC2				:BOOL;	(* Diagnosis μC2 - Value 204 - External supply 24 V output 2 *)
	
END_STRUCT
END_TYPE
(* End *)

// ---- DUTs/TwinSAFE/TwinSAFE_Connection/EK1914/ST_TsDiagObjectsEK1914.TcDUT
TYPE ST_TsDiagObjectsEK1914 :
(*******************************************************************************************************
Description			:	Index 16#800E Diagnostic objects
Supported terminals : 	EK1914
Documentation 		:	EK1914 TwinSAFE input/output terminal with 2 fail-safe inputs and 2 fail-safe outputs
Version/Date 		:	V1.2.0/08.03.2016
********************************************************************************************************)
STRUCT
	
	nDummyData1								:ARRAY[0..8] OF UINT;

(* Sensor test error *)
	nSensorTestError						:UINT;

(* Error during two channel evaluation *)
	nDuringTwoChannelEvaluationError		:UINT;

(* Error in the safety mat operating mode: input pair disagree *)
	nMatModeInputPairDisagreeError			:UINT;

(* Error in the safety mat operating mode: external supply *)
	nMatModeExternalSupplyError				:UINT;

(* Diagnosis μC1 *)
	nDiagnosisMicroC1						:UINT;

(* Diagnosis μC2 *)
	nDiagnosisMicroC2						:UINT;

	nDummyData2								:ARRAY[0..48] OF UINT;

END_STRUCT
END_TYPE
(* End *)

// ---- DUTs/TwinSAFE/TwinSAFE_Connection/EK1914/ST_TsSlaveInfoEK1914.TcDUT
TYPE ST_TsSlaveInfoEK1914 :
STRUCT

(* act_EcSlaveIdentify *)
	sEcSlaveType							:STRING(15);
	sEcSlaveName							:STRING(31) := '';
	bSlaveIdentify							:BOOL;
	bSlaveTypeError							:BOOL;
	
(* act_Signals *)
	bChannel1In								:BOOL;							
	bChannel2In								:BOOL;
	bChannel1Out							:BOOL;
	bChannel2Out							:BOOL;

(* act_ConnectionState *)
	sState									:STRING;
	
(* act_ConnectionDiag *)
	sDiag									:STRING;
	sFault									:STRING;						(* FailSafe Error (Hardware)*)
	bError									:BOOL;							(* TwinSAFE-Error *)
	
(* act_ReadDiagObjects *)
	stSlaveTemp								:ST_TsSlave2Temp;
	bIntTempWarning1						:BOOL;							(* Temperature warning: T1 *)
	bIntTempWarning2						:BOOL;							(* Temperature warning: T2 *)
	stTsDiagObjectsBitsEK1914				:ST_TsDiagObjectsBitsEK1914;

END_STRUCT
END_TYPE
(*End*)

// ---- DUTs/TwinSAFE/TwinSAFE_Connection/EK1960/ST_TsConnectionInfoEK1960.TcDUT
TYPE ST_TsConnectionInfoEK1960 :
(*******************************************************************************************************
Description			:	Connection information data of EtherCAT Slaves with 12 byte safe data   
Supported terminals : 	EK1960
Date 				:	04.11.2018
********************************************************************************************************)
STRUCT

	nState  								:USINT;
	nDiag 	 								:USINT;
	
	nInOutSafeDataByte1	 					:BYTE;
	nInOutSafeDataByte2	 					:BYTE;
	nInOutSafeDataByte3	 					:BYTE;
	nInOutSafeDataByte4 					:BYTE;
	nInOutSafeDataByte5 					:BYTE;
	nInOutSafeDataByte6 					:BYTE;
	nInOutSafeDataByte7 					:BYTE;
	nInOutSafeDataByte8 					:BYTE;
	nInOutSafeDataByte9 					:BYTE;
	nInOutSafeDataByte10					:BYTE;
	nInOutSafeDataByte11					:BYTE;
	nInOutSafeDataByte12					:BYTE;

END_STRUCT
END_TYPE
(* End *)

// ---- DUTs/TwinSAFE/TwinSAFE_Connection/EK1960/ST_TsDeviceInfoDataEK1960.TcDUT
TYPE ST_TsDeviceInfoDataEK1960 :
(*******************************************************************************************************
Description			:	EtherCAT master terminals device info controller
Supported terminals : 	EL1918 / EK1960
Date 				:	25.05.2018
********************************************************************************************************)
STRUCT
	nVoltageC						:UINT;	(* Voltage controller [mV] *)
	nTemperatureC					:INT;	(* Temperature controller [°C] *)
	nFirmwareCrcC					:UINT;	(* CRC Firmware *)
	nVendorDataCrcC					:UINT;	(* CRC Vendor Data *)	
END_STRUCT
END_TYPE
(* End *)

// ---- DUTs/TwinSAFE/TwinSAFE_Connection/EK1960/ST_TsDiagObjectsEK1960.TcDUT
TYPE ST_TsDiagObjectsEK1960 :
(*******************************************************************************************************
Description			:	Index 16#800E Diagnostic objects
Supported terminals : 	EK1960
Documentation 		:	EK1960 TwinSAFE compact-controller
Version/Date 		:	V1.5.3/21.01.2019
********************************************************************************************************)
STRUCT

	nDummyData1								:ARRAY[0..8] OF UINT;

(* Sensor test error *)
	nSensorTestError						:UINT;

(* Error during two channel evaluation *)
	nDuringTwoChannelEvaluationError		:UINT;

(* Error in the safety mat operating mode: input pair disagree *)
	nMatModeInputPairDisagreeError			:UINT;

(* Error in the safety mat operating mode: external supply *)
	nMatModeExternalSupplyError				:UINT;

	nDummyData2								:ARRAY[0..2] OF UINT;

END_STRUCT
END_TYPE
(* End *)

// ---- DUTs/TwinSAFE/TwinSAFE_Connection/EK1960/ST_TsSlaveInfoEK1960.TcDUT
TYPE ST_TsSlaveInfoEK1960 :
STRUCT
	
(* act_EcSlaveIdentify *)
	sEcSlaveType							:STRING(15);
	bSlaveIdentify							:BOOL;
	bSlaveTypeError							:BOOL;
	
	sEcSlaveName							:STRING(31) := '';

	stTsSlaveAddress 						:ST_TsSlaveAddressCRC;
	bSlaveAddressOk							:BOOL;
	
	nEcSlaveFSoEAddr						:UINT;
	nEcSlaveSerialNumber					:UDINT;
	nEcProjectCrc							:UINT;

(* act_Signals *)
	bFSINModule1Channel1		   			:BOOL;
	bFSINModule1Channel2		   			:BOOL;
	bFSINModule1ModuleFault		   			:BOOL;
	bFSINModule1ErrAck			   			:BOOL;

	bFSINModule2Channel1		   			:BOOL;
	bFSINModule2Channel2		   			:BOOL;
	bFSINModule2ModuleFault		   			:BOOL;
	bFSINModule2ErrAck			   			:BOOL;

	bFSINModule3Channel1		   			:BOOL;
	bFSINModule3Channel2		   			:BOOL;
	bFSINModule3ModuleFault		   			:BOOL;
	bFSINModule3ErrAck			   			:BOOL;

	bFSINModule4Channel1		   			:BOOL;
	bFSINModule4Channel2		   			:BOOL;
	bFSINModule4ModuleFault		   			:BOOL;
	bFSINModule4ErrAck			   			:BOOL;

	bFSINModule5Channel1		   			:BOOL;
	bFSINModule5Channel2		   			:BOOL;
	bFSINModule5ModuleFault		   			:BOOL;
	bFSINModule5ErrAck			   			:BOOL;

	bFSINModule6Channel1		   			:BOOL;
	bFSINModule6Channel2		  			:BOOL;
	bFSINModule6ModuleFault		   			:BOOL;
	bFSINModule6ErrAck			   			:BOOL;

	bFSINModule7Channel1		   			:BOOL;
	bFSINModule7Channel2		   			:BOOL;
	bFSINModule7ModuleFault		   			:BOOL;
	bFSINModule7ErrAck			   			:BOOL;

	bFSINModule8Channel1		   			:BOOL;
	bFSINModule8Channel2		  			:BOOL;
	bFSINModule8ModuleFault		   			:BOOL;
	bFSINModule8ErrAck			   			:BOOL;

	bFSINModule9Channel1		   			:BOOL;
	bFSINModule9ModuleFault1	   			:BOOL;
	bFSINModule9ErrAck1			   			:BOOL;
	bFSINModule9Channel2		   			:BOOL;
	bFSINModule9ModuleFault2	   			:BOOL;
	bFSINModule9ErrAck2			   			:BOOL;

	bFSINModule10Channel1		   			:BOOL;
	bFSINModule10ModuleFault1	   			:BOOL;
	bFSINModule10ErrAck1		   			:BOOL;
	bFSINModule10Channel2		   			:BOOL;
	bFSINModule10ModuleFault2	  			:BOOL;
	bFSINModule10ErrAck2		   			:BOOL;

	(* Outputs *)	
	bFSOUTModule1Channel1		   			:BOOL;
	bFSOUTModule1Channel2		   			:BOOL;
	bFSOUTModule1Channel3		   			:BOOL;
	bFSOUTModule1Channel4		   			:BOOL;
	bFSOUTModule1ModuleFault			  	:BOOL;
	bFSOUTModule1ErrAck			   			:BOOL;
	
	bFSOUTModule2Channel1		   			:BOOL;
	bFSOUTModule2Channel2		   			:BOOL;
	bFSOUTModule2Channel3		   			:BOOL;
	bFSOUTModule2Channel4		   			:BOOL;
	bFSOUTModule2ModuleFault			   	:BOOL;
	bFSOUTModule2ErrAck			 			:BOOL;
	
	bFSOUTModule3Channel1		   			:BOOL;
	bFSOUTModule3Channel2		   			:BOOL;
	bFSOUTModule3Channel3		   			:BOOL;
	bFSOUTModule3Channel4		   			:BOOL;
	bFSOUTModule3ModuleFault	   			:BOOL;
	bFSOUTModule3ErrAck			   			:BOOL;
	
	bFSOUTModule4Channel1		   			:BOOL;
	bFSOUTModule4Channel2		   			:BOOL;
	bFSOUTModule4Channel3		   			:BOOL;
	bFSOUTModule4Channel4		   			:BOOL;
	bFSOUTModule4ModuleFault	   			:BOOL;
	bFSOUTModule4ErrAck			   			:BOOL;
	
	bFSOUTModule5Channel1		   			:BOOL;
	bFSOUTModule5Channel2		   			:BOOL;
	bFSOUTModule5Channel3		  			:BOOL;
	bFSOUTModule5Channel4		   			:BOOL;
	bFSOUTModule5ModuleFault	   			:BOOL;
	bFSOUTModule5ErrAck			  			:BOOL;
	
	bFSOUTModule6Channel1		   			:BOOL;
	bFSOUTModule6Channel2		   			:BOOL;
	bFSOUTModule6Channel3		   			:BOOL;
	bFSOUTModule6Channel4		   			:BOOL;
	bFSOUTModule6ModuleFault	   			:BOOL;
	bFSOUTModule6ErrAck			   			:BOOL;
	
	bFSOUTRelaisModuleChannel1	   			:BOOL;
	bFSOUTRelaisModuleChannel2	   			:BOOL;
	bFSOUTRelaisModuleChannel3	   			:BOOL;
	bFSOUTRelaisModuleChannel4	   			:BOOL;
	bFSOUTRelaisModuleFault		   			:BOOL;
	bFSOUTRelaisModuleErrAck	   			:BOOL;
	
(* act_ConnectionDiag *)
	sDiag									:STRING;
	sFault									:STRING;						(* FailSafe Error (Hardware)*)
	bError									:BOOL;							(* TwinSAFE-Error *)
	
(* act_ConnectionState *)
	sState									:STRING;
	
	(* act_ReadDiagObjects *)
	stSlaveTemp								:ST_TsSlave2Temp;
	bIntTempWarning1						:BOOL;							(* Temperature warning: T1 *)
	bIntTempWarning2						:BOOL;							(* Temperature warning: T2 *)
	stTsDiagObjectsBitsEK1960				:ARRAY[1..2] OF ST_TsDeviceInfoDataEK1960;
	
END_STRUCT
END_TYPE
(*End*)

// ---- DUTs/TwinSAFE/TwinSAFE_Connection/EL1918/ST_TsConnectionInfoEL1918.TcDUT
{attribute 'pack_mode' := '0'}
TYPE ST_TsConnectionInfoEL1918 :
(*******************************************************************************************************
Description			:	Connection information data of EtherCAT Slaves with 2 byte input and 1 byte output safe data  
Supported terminals : 	EL1918 (asIO-terminal
Date 				:	04.11.2018
********************************************************************************************************)
STRUCT

	nState  								:USINT;
	nDiag 	 								:USINT;
	nInOutSafeDataByte1						:BYTE;
	nInOutSafeDataByte2						:BYTE;
	nInOutSafeDataByte3						:BYTE;

END_STRUCT
END_TYPE
(* End *)

// ---- DUTs/TwinSAFE/TwinSAFE_Connection/EL1918/ST_TsDeviceInfoDataEL1918.TcDUT
TYPE ST_TsDeviceInfoDataEL1918 :
(*******************************************************************************************************
Description			:	EtherCAT master terminals device info controller
Supported terminals : 	EL1918
Date 				:	25.05.2018
********************************************************************************************************)
STRUCT
	nVoltageC						:UINT;	(* Voltage controller [mV] *)
	nTemperatureC					:INT;	(* Temperature controller [°C] *)
	nFirmwareCrcC					:UINT;	(* CRC Firmware *)
	nVendorDataCrcC					:UINT;	(* CRC Vendor Data *)	
END_STRUCT
END_TYPE
(* End *)

// ---- DUTs/TwinSAFE/TwinSAFE_Connection/EL1918/ST_TsDiagObjectsEL1918.TcDUT
TYPE ST_TsDiagObjectsEL1918 :
(*******************************************************************************************************
Description			:	Index 16#800E Diagnostic objects
Supported terminals : 	EL1904, EL1918
Documentation 		:	EL1918, TwinSAFE input terminal with 8 fail-safe inputs
Version/Date 		:	V1.5.2/02.10.2015
********************************************************************************************************)
STRUCT

	nDummyData1								:ARRAY[0..8] OF UINT;

(* Sensor test error *)
	nSensorTestError						:UINT;

(* Error during two channel evaluation *)
	nDuringTwoChannelEvaluationError		:UINT;

(* Error in the safety mat operating mode: input pair disagree *)
	nMatModeInputPairDisagreeError			:UINT;

(* Error in the safety mat operating mode: external supply *)
	nMatModeExternalSupplyError				:UINT;

	nDummyData2								:ARRAY[0..2] OF UINT;

END_STRUCT
END_TYPE
(* End *)

// ---- DUTs/TwinSAFE/TwinSAFE_Connection/EL1918/ST_TsSlaveInfoEL1918.TcDUT
TYPE ST_TsSlaveInfoEL1918 :
STRUCT

(* act_EcSlaveIdentify *)
	sEcSlaveType							:STRING(15);
	sEcSlaveName							:STRING(31) := '';
	bSlaveIdentify							:BOOL;
	bSlaveTypeError							:BOOL;
	{attribute 'displaymode':='hex'}
	nEcProjectCrc							:UINT;

	stTsSlaveAddress 						:ST_TsSlaveAddressCRC;
	bSlaveAddressOk							:BOOL;
	
	nEcSlaveFSoEAddr						:UINT;
	nEcSlaveSerialNumber					:UDINT;
	
(* act_ConnectionState *)
	sState									:STRING;
	
(* act_ConnectionDiag *)
	sDiag									:STRING;
	sFault									:STRING;						(* FailSafe Error (Hardware)*)
	bError									:BOOL;							(* TwinSAFE-Error *)
	
(* act_ReadDiagObjects *)
	stSlaveTemp								:ST_TsSlave2Temp;
	bIntTempWarning1						:BOOL;							(* Temperature warning: T1 *)
	bIntTempWarning2						:BOOL;							(* Temperature warning: T2 *)
	stTsDiagObjectsBitsEL1918				:ARRAY[1..2] OF ST_TsDeviceInfoDataEL1918;	

(* act_Signals *)
	bChannel1								:BOOL;							
	bChannel1ModuleFault					:BOOL;							
	bChannel1ErrAck							:BOOL;
	
	bChannel2								:BOOL;
	bChannel2ModuleFault					:BOOL;							
	bChannel2ErrAck							:BOOL;

	bChannel3								:BOOL;
	bChannel3ModuleFault					:BOOL;							
	bChannel3ErrAck							:BOOL;

	bChannel4								:BOOL;
	bChannel4ModuleFault					:BOOL;							
	bChannel4ErrAck							:BOOL;

	bChannel5								:BOOL;
	bChannel5ModuleFault					:BOOL;							
	bChannel5ErrAck							:BOOL;

	bChannel6								:BOOL;
	bChannel6ModuleFault					:BOOL;							
	bChannel6ErrAck							:BOOL;

	bChannel7								:BOOL;
	bChannel7ModuleFault					:BOOL;							
	bChannel7ErrAck							:BOOL;

	bChannel8								:BOOL;
	bChannel8ModuleFault					:BOOL;							
	bChannel8ErrAck							:BOOL;

END_STRUCT
END_TYPE
(*End*)

// ---- DUTs/TwinSAFE/TwinSAFE_Connection/EL2911/ST_TsConnectionInfoEL2911.TcDUT
TYPE ST_TsConnectionInfoEL2911 :
(*******************************************************************************************************
Description			:	Connection information data of EtherCAT Slaves with 2 byte input and 2 byte output safe data  
Supported terminals : 	EP1957, EL2911
Date 				:	04.11.2018
********************************************************************************************************)
STRUCT

	nState  								:USINT;
	nDiag 	 								:USINT;
	nInOutSafeDataByte1						:BYTE;
	nInOutSafeDataByte2						:BYTE;

END_STRUCT
END_TYPE
(* End *)

// ---- DUTs/TwinSAFE/TwinSAFE_Connection/EL2911/ST_TsDeviceInfoDataEL2911.TcDUT
TYPE ST_TsDeviceInfoDataEL2911 :
(*******************************************************************************************************
Description			:	EtherCAT master terminals device info controller
Supported terminals : 	EL2911
Date 				:	25.05.2018
********************************************************************************************************)
STRUCT
	nVoltageC						:UINT;	(* Voltage controller [mV] *)
	nTemperatureC					:INT;	(* Temperature controller [°C] *)
	nFirmwareCrcC					:UINT;	(* CRC Firmware *)
	nVendorDataCrcC					:UINT;	(* CRC Vendor Data *)	
END_STRUCT
END_TYPE
(* End *)

// ---- DUTs/TwinSAFE/TwinSAFE_Connection/EL2911/ST_TsDiagObjectsEL2911.TcDUT
TYPE ST_TsDiagObjectsEL2911 :
(*******************************************************************************************************
Description			:	Index 16#800E Diagnostic objects
Supported terminals : 	EL1904, EL2911
Documentation 		:	EL2911 TwinSAFE potential supply terminal with 4 fail-safe inputs and 1 fail-safe output
Version/Date 		:	V1.5.2/02.10.2015
********************************************************************************************************)
STRUCT

	nDummyData1								:ARRAY[0..8] OF UINT;

(* Sensor test error *)
	nSensorTestError						:UINT;

(* Error during two channel evaluation *)
	nDuringTwoChannelEvaluationError		:UINT;

(* Error in the safety mat operating mode: input pair disagree *)
	nMatModeInputPairDisagreeError			:UINT;

(* Error in the safety mat operating mode: external supply *)
	nMatModeExternalSupplyError				:UINT;

	nDummyData2								:ARRAY[0..2] OF UINT;

END_STRUCT
END_TYPE
(* End *)

// ---- DUTs/TwinSAFE/TwinSAFE_Connection/EL2911/ST_TsSlaveInfoEL2911.TcDUT
TYPE ST_TsSlaveInfoEL2911 :
STRUCT
	
(* act_EcSlaveIdentify *)
	sEcSlaveType							:STRING(15);
	sEcSlaveName							:STRING(31) := '';
	bSlaveIdentify							:BOOL;
	bSlaveTypeError							:BOOL;
	{attribute 'displaymode':='hex'}
	nEcProjectCrc							:UINT;
	
	stTsSlaveAddress 						:ST_TsSlaveAddressCRC;
	bSlaveAddressOk							:BOOL;
	
	nEcSlaveFSoEAddr						:UINT;
	nEcSlaveSerialNumber					:UDINT;
	
(* act_ConnectionState *)
	sState									:STRING;
	
(* act_ConnectionDiag *)
	sDiag									:STRING;
	sFault									:STRING;						(* FailSafe Error (Hardware)*)
	bError									:BOOL;							(* TwinSAFE-Error *)
	
(* act_ReadDiagObjects *)
	stSlaveTemp								:ST_TsSlave2Temp;
	bIntTempWarning1						:BOOL;							(* Temperature warning: T1 *)
	bIntTempWarning2						:BOOL;							(* Temperature warning: T2 *)
	stTsDiagObjectsBitsEL2911				:ARRAY[1..2] OF ST_TsDeviceInfoDataEL2911;
	
(* act_Signals *)
	(* Inputs *)
	bFSINChannel1         					:BOOL;
	bFSINChannel2        					:BOOL;
	bFSINChannel3        					:BOOL;
	bFSINChannel4        					:BOOL;
	bFSINModuleFault    					:BOOL;
	bFSINModuleErrAck 						:BOOL;
	
	(* Outputs *)
	bFSOUTChannel1     						:BOOL;
	bFSOUTModuleFault   					:BOOL;
	bFSOUTModuleErrAck	   					:BOOL;

END_STRUCT
END_TYPE
(*End*)

// ---- DUTs/TwinSAFE/TwinSAFE_Connection/EL2912/ST_TsConnectionInfoEL2912.TcDUT
TYPE ST_TsConnectionInfoEL2912 :
(*******************************************************************************************************
Description			:	Connection information data of EtherCAT Slaves with 2 byte input and 2 byte output safe data  
Supported terminals : 	EL2912
Date 				:	20.12.2021
********************************************************************************************************)
STRUCT

	nState  								:USINT;
	nDiag 	 								:USINT;
	nInOutSafeDataByte1						:BYTE;
	nInOutSafeDataByte2						:BYTE;

END_STRUCT
END_TYPE
(* End *)

// ---- DUTs/TwinSAFE/TwinSAFE_Connection/EL2912/ST_TsDeviceInfoDataEL2912.TcDUT
TYPE ST_TsDeviceInfoDataEL2912 :
(*******************************************************************************************************
Description			:	EtherCAT master terminals device info controller
Supported terminals : 	EL2912
Date 				:	20.12.2021
********************************************************************************************************)
STRUCT
	nVoltageC						:UINT;	(* Voltage controller [mV] *)
	nTemperatureC					:INT;	(* Temperature controller [°C] *)
	nFirmwareCrcC					:UINT;	(* CRC Firmware *)
	nVendorDataCrcC					:UINT;	(* CRC Vendor Data *)	
END_STRUCT
END_TYPE
(* End *)

// ---- DUTs/TwinSAFE/TwinSAFE_Connection/EL2912/ST_TsDiagObjectsEL2912.TcDUT
TYPE ST_TsDiagObjectsEL2912 :
(*******************************************************************************************************
Description			:	Index 16#800E Diagnostic objects
Supported terminals : 	EL2912
Documentation 		:	EL2912 TwinSAFE potential supply terminal with 4 fail-safe inputs and 1 fail-safe output
Version/Date 		:	20.12.2021
********************************************************************************************************)
STRUCT

	nDummyData1								:ARRAY[0..8] OF UINT;

(* Sensor test error *)
	nSensorTestError						:UINT;

(* Error during two channel evaluation *)
	nDuringTwoChannelEvaluationError		:UINT;

(* Error in the safety mat operating mode: input pair disagree *)
	nMatModeInputPairDisagreeError			:UINT;

(* Error in the safety mat operating mode: external supply *)
	nMatModeExternalSupplyError				:UINT;

	nDummyData2								:ARRAY[0..2] OF UINT;

END_STRUCT
END_TYPE
(* End *)

// ---- DUTs/TwinSAFE/TwinSAFE_Connection/EL2912/ST_TsSlaveInfoEL2912.TcDUT
TYPE ST_TsSlaveInfoEL2912 :
STRUCT
	
(* act_EcSlaveIdentify *)
	sEcSlaveType							:STRING(15);
	sEcSlaveName							:STRING(31) := '';
	bSlaveIdentify							:BOOL;
	bSlaveTypeError							:BOOL;
	{attribute 'displaymode':='hex'}
	nEcProjectCrc							:UINT;
	
	stTsSlaveAddress 						:ST_TsSlaveAddressCRC;
	bSlaveAddressOk							:BOOL;
	
	nEcSlaveFSoEAddr						:UINT;
	nEcSlaveSerialNumber					:UDINT;
	
(* act_ConnectionState *)
	sState									:STRING;
	
(* act_ConnectionDiag *)
	sDiag									:STRING;
	sFault									:STRING;						(* FailSafe Error (Hardware)*)
	bError									:BOOL;							(* TwinSAFE-Error *)
	
(* act_ReadDiagObjects *)
	stSlaveTemp								:ST_TsSlave2Temp;
	bIntTempWarning1						:BOOL;							(* Temperature warning: T1 *)
	bIntTempWarning2						:BOOL;							(* Temperature warning: T2 *)
	stTsDiagObjectsBitsEL2912				:ARRAY[1..2] OF ST_TsDeviceInfoDataEL2912;
	
(* act_Signals *)	
	(* Outputs *)
	bFSOUTChannel1     						:BOOL;
	bFSOUTChannel2     						:BOOL;
	bFSOUTModule1Fault   					:BOOL;
	bFSOUTModule2Fault   					:BOOL;
	bFSOUTModule1ErrAck	   					:BOOL;
	bFSOUTModule2ErrAck	   					:BOOL;

END_STRUCT
END_TYPE
(*End*)

// ---- DUTs/TwinSAFE/TwinSAFE_Connection/EL3214/ST_TsConnectionInfoEL3214.TcDUT
TYPE ST_TsConnectionInfoEL3214 :
(*******************************************************************************************************
Description			:	Connection information data of EtherCAT Slave EL3214-0090 with 4 analog inputs  
Supported terminals : 	EL3214-0090
Date 				:	01.12.2016
********************************************************************************************************)
STRUCT

	nState  								:USINT;
	nDiag 	 								:USINT;
	nInSafeDataValue1						:INT;
	nInSafeDataValue2						:INT;
	nInSafeDataValue3						:INT;
	nInSafeDataValue4						:INT;

END_STRUCT
END_TYPE
(* End *)

// ---- DUTs/TwinSAFE/TwinSAFE_Connection/EL3214/ST_TsSlaveInfoEL3214.TcDUT
TYPE ST_TsSlaveInfoEL3214 :
STRUCT
	
(* act_EcSlaveIdentify *)
	sEcSlaveType							:STRING(15);
	sEcSlaveName							:STRING(31) := '';
	bSlaveIdentify							:BOOL;
	bSlaveTypeError							:BOOL;
	
(* act_ConnectionState *)
	sState									:STRING;
	
(* act_ConnectionDiag *)
	sDiag									:STRING;
	sFault									:STRING;						(* FailSafe Error (Hardware)*)
	bError									:BOOL;							(* TwinSAFE-Error *)	

(* act_Signals *)
	nInSafeDataValue1						:UINT;
	nInSafeDataValue2						:INT;
	nInSafeDataValue3						:INT;
	nInSafeDataValue4						:INT;

END_STRUCT
END_TYPE
(*End*)

// ---- DUTs/TwinSAFE/TwinSAFE_Connection/EL5021/ST_TsConnectionInfoEL5021.TcDUT
TYPE ST_TsConnectionInfoEL5021 :
(*******************************************************************************************************
Description			:	Connection information data of EtherCAT Slave EL5021-0090 with 1 counter (1 Vss) input 
Supported terminals : 	EL5021-0090
Date 				:	01.12.2016
********************************************************************************************************)
STRUCT

	nState  								:USINT;
	nDiag 	 								:USINT;
	nInSafeDataCounterValue					:UDINT;
	nInSafeDataFrequencyValue				:DINT;

END_STRUCT
END_TYPE
(* End *)

// ---- DUTs/TwinSAFE/TwinSAFE_Connection/EL5021/ST_TsSlaveInfoEL5021.TcDUT
TYPE ST_TsSlaveInfoEL5021 :
STRUCT

(* act_EcSlaveIdentify *)
	sEcSlaveType							:STRING(15);
	sEcSlaveName							:STRING(31) := '';
	bSlaveIdentify							:BOOL;
	bSlaveTypeError							:BOOL;

(* act_ConnectionState *)
	sState									:STRING;
	
(* act_ConnectionDiag *)
	sDiag									:STRING;
	sFault									:STRING;						(* FailSafe Error (Hardware)*)
	bError									:BOOL;							(* TwinSAFE-Error *)	
	
(* act_Signals *)
	nInSafeDataCounterValue					:UDINT;
	nInSafeDataFrequencyValue				:DINT;
//	nInSafeDataFrequencyValue16Bit			:INT;

END_STRUCT
END_TYPE
(*End*)

// ---- DUTs/TwinSAFE/TwinSAFE_Connection/EL6900/ST_TsHardwareDiagC.TcDUT
TYPE ST_TsHardwareDiagC :
(*******************************************************************************************************
Description			:	EtherCAT master terminals hardware diagnosis controller
Supported terminals : 	EL6900
Date 				:	25.05.2018
********************************************************************************************************)
STRUCT

	nTemperatureC1					:INT;	(* Temperature controller 1 [°C] *)
	nTemperatureC2					:INT;	(* Temperature controller 2 [°C] *)
	nVoltageC1						:UINT;	(* Voltage controller 1 [mV] *)
	nVoltageC2						:UINT;	(* Voltage controller 2 [mV] *)
	
END_STRUCT
END_TYPE
(* End *)

// ---- DUTs/TwinSAFE/TwinSAFE_Connection/EL6900/ST_TsSlaveInfoEL6900.TcDUT
TYPE ST_TsSlaveInfoEL6900 :
STRUCT
	
(* act_EcSlaveIdentify *)
	sEcSlaveType							:STRING(15);
	sEcSlaveName							:STRING(31) := '';
	bSlaveIdentify							:BOOL;
	bSlaveTypeError							:BOOL;
	{attribute 'displaymode':='hex'}
	nEcSlaveProjectCRC						:UINT;
	
	stTsSlaveAddress 						:ST_TsSlaveAddressCRC;
	bSlaveAddressOk							:BOOL;
	
	nEcSlaveFSoEAddr						:UINT;
	nEcSlaveSerialNumber					:UDINT;
	
(* act_ReadDiagObjects *)
	stHardwareDiagC							:ST_TsHardwareDiagC;
	bIntTempWarning1						:BOOL;							(* Temperature warning: T1 *)
	bIntTempWarning2						:BOOL;							(* Temperature warning: T2 *)

END_STRUCT
END_TYPE
(*End*)

// ---- DUTs/TwinSAFE/TwinSAFE_Connection/EP1957/ST_TsConnectionInfoEP1957.TcDUT
TYPE ST_TsConnectionInfoEP1957 :
(*******************************************************************************************************
Description			:	Connection information data of EtherCAT Slaves with 2 byte input and 2 byte output safe data  
Supported terminals : 	EP1957
Date 				:	04.11.2018
********************************************************************************************************)
STRUCT

	nState  								:USINT;
	nDiag 	 								:USINT;
	nInOutSafeDataByte1						:BYTE;
	nInOutSafeDataByte2						:BYTE;
	nInOutSafeDataByte3						:BYTE;
	nInOutSafeDataByte4						:BYTE;

END_STRUCT
END_TYPE
(* End *)

// ---- DUTs/TwinSAFE/TwinSAFE_Connection/EP1957/ST_TsDeviceInfoDataEP1957.TcDUT
TYPE ST_TsDeviceInfoDataEP1957 :
(*******************************************************************************************************
Description			:	EtherCAT master terminals device info controller
Supported terminals : 	EL1918, EP1957
Date 				:	25.05.2018
********************************************************************************************************)
STRUCT
	nVoltageC						:UINT;	(* Voltage controller [mV] *)
	nTemperatureC					:INT;	(* Temperature controller [°C] *)
	nFirmwareCrcC					:UINT;	(* CRC Firmware *)
	nVendorDataCrcC					:UINT;	(* CRC Vendor Data *)	
END_STRUCT
END_TYPE
(* End *)

// ---- DUTs/TwinSAFE/TwinSAFE_Connection/EP1957/ST_TsDiagObjectsEP1957.TcDUT
TYPE ST_TsDiagObjectsEP1957 :
(*******************************************************************************************************
Description			:	Index 16#800E Diagnostic objects
Supported terminals : 	EL1904, EP1957
Documentation 		:	EP1957 TwinSAFE input terminal with 8 fail-safe inputs
Version/Date 		:	V1.5.2/02.10.2015
********************************************************************************************************)
STRUCT

	nDummyData1								:ARRAY[0..8] OF UINT;

(* Sensor test error *)
	nSensorTestError						:UINT;

(* Error during two channel evaluation *)
	nDuringTwoChannelEvaluationError		:UINT;

(* Error in the safety mat operating mode: input pair disagree *)
	nMatModeInputPairDisagreeError			:UINT;

(* Error in the safety mat operating mode: external supply *)
	nMatModeExternalSupplyError				:UINT;

	nDummyData2								:ARRAY[0..2] OF UINT;

END_STRUCT
END_TYPE
(* End *)

// ---- DUTs/TwinSAFE/TwinSAFE_Connection/EP1957/ST_TsSlaveInfoEP1957.TcDUT
TYPE ST_TsSlaveInfoEP1957 :
STRUCT
	
(* act_EcSlaveIdentify *)
	sEcSlaveType							:STRING(15);
	sEcSlaveName							:STRING(31) := '';
	bSlaveIdentify							:BOOL;
	bSlaveTypeError							:BOOL;
	{attribute 'displaymode':='hex'}
	nEcProjectCrc							:UINT;
	
	stTsSlaveAddress 						:ST_TsSlaveAddressCRC;
	bSlaveAddressOk							:BOOL;
	
	nEcSlaveFSoEAddr						:UINT;
	nEcSlaveSerialNumber					:UDINT;
	
(* act_ConnectionState *)
	sState									:STRING;
	
(* act_ConnectionDiag *)
	sDiag									:STRING;
	sFault									:STRING;						(* FailSafe Error (Hardware)*)
	bError									:BOOL;							(* TwinSAFE-Error *)
	
(* act_ReadDiagObjects *)
	stSlaveTemp								:ST_TsSlave2Temp;
	bIntTempWarning1						:BOOL;							(* Temperature warning: T1 *)
	bIntTempWarning2						:BOOL;							(* Temperature warning: T2 *)
	stTsDiagObjectsBitsEP1957				:ARRAY[1..2] OF ST_TsDeviceInfoDataEP1957;

(* act_Signals *)
	(* Inputs *)
	bFSINChannel1         					:BOOL;
	bFSINChannel2        					:BOOL;
	bFSINModule1Fault    					:BOOL;
	bFSINModule1ErrAck  					:BOOL;

	bFSINChannel3        					:BOOL;
	bFSINChannel4        					:BOOL;
	bFSINModule2Fault    					:BOOL;
	bFSINModule2ErrAck   					:BOOL;

	bFSINChannel5        					:BOOL;
	bFSINChannel6        					:BOOL;
	bFSINModule3Fault    					:BOOL;
	bFSINModule3ErrAck   					:BOOL;

	bFSINChannel7        					:BOOL;
	bFSINChannel8        					:BOOL;
	bFSINModule4Fault    					:BOOL;
	bFSINModule4ErrAck   					:BOOL;
                   
	(* Outputs *)
	bFSOUTChannel1     						:BOOL;
	bFSOUTModule1Fault   					:BOOL;
	bFSOUTModule1ErrAck	   					:BOOL;

	bFSOUTChannel2     						:BOOL;
	bFSOUTModule2Fault 	   					:BOOL;
	bFSOUTModule2ErrAck	   					:BOOL;

	bFSOUTChannel3     						:BOOL;
	bFSOUTModule3Fault 	   					:BOOL;
	bFSOUTModule3ErrAck	   					:BOOL;

	bFSOUTChannel4     						:BOOL;
	bFSOUTModule4Fault 	   					:BOOL;
	bFSOUTModule4ErrAck					   	:BOOL;

END_STRUCT
END_TYPE
(*End*)

// ---- GVLs/GVL.TcGVL
{attribute 'qualified_only'}
VAR_GLOBAL
	//Thermocouple
	nTemp AT %I*: INT;
	bSwOn AT %I*: BOOL; //Self reset
	bSwOff AT %I*: BOOL; //Self reset
	bLight AT %Q*: BOOL;
	bFan AT %Q*: BOOL;
	
	//Power measurement
	fIL1 AT %I*: REAL; //RMS Current
	fUL1 AT %I*: REAL; //RMS Voltage
	fActivePower AT %I*: REAL; //Active Power
	fcosphi1 AT %I*: REAL; //Phase angle
	fFrequency AT %I*: REAL; //Frequency
	
	//Motor drive
	stAxis1: AXIS_REF;
	bButtonFw AT %I*: BOOL:=FALSE; //Self reset
	bButtonBw AT %I*: BOOL:=FALSE; //Self reset
	bButtonHalt AT %I*: BOOL:=FALSE; //Self reset
	bButtonAuto AT %I*: BOOL; //Latch
	
	//VFD Modbus RTU
	bRunVfd AT %I*: BOOL;
	bStopVfd AT %I*: BOOL;
	bEnable: BOOL; //Self reset
	bDisable: BOOL; //Self reset
	bReverseMotor: BOOL; //Self reset
	bSetMotorFrequency: BOOL; //Self reset
	
	// Bit 0 and Bit 1 declaration
	bModbusCoilBit0 : BOOL;
	bModbusCoilBit1 : BOOL;
	
	// Virtual toggle buttons for write values using MODBUS RTU
	bExecuteWriteCoils: BOOL;
	bExecuteWriteRegs0: BOOL;
	bExecuteWriteSingleRegForHmi: BOOL;
	//bExecuteWriteRegs1: BOOL;

	// Input STRING from HMI, MAXIMUM 20 characters
	sInputFromHMI: STRING(20):='Beckhoff VN';		

	//Constant value for testing, used for EL2596
	bLedEnable AT %Q*:BOOL:=TRUE;
	bLedOutput AT %Q*:BOOL:=TRUE;
	bOutputCurrent AT %Q*: UINT:=300;
	
	// Constant value for EL2809 controlling strobe
	bLedEnableEL2xxx AT %Q*:BOOL;
	bLedEnableVirtualInputButton: BOOL; 	

	// Loadcell scaling variables
	uLoadCellRawValue AT %I*: DINT;
	uLoadCellScaledValue: REAL;
	
	// Output signal variables for sneumatic valves 
	bValve1 AT %Q*:BOOL;
	bValve2 AT %Q*:BOOL;
	bValve3 AT %Q*:BOOL;
	bValve4 AT %Q*:BOOL;
	bValve5 AT %Q*:BOOL;
	bValve6 AT %Q*:BOOL;
	bVirtualToggleButton1:BOOL;
	bVirtualToggleButton2:BOOL;
	bVirtualToggleButton3:BOOL;
	bVirtualToggleButton4:BOOL;
	bVirtualToggleButton5:BOOL;
	bVirtualToggleButton6:BOOL;
	
	// TwinSAFE declaration
	(*bSafeRun AT %Q*:BOOL;
	bSafeAck AT %Q*:BOOL;
	bSafeFBErr AT %I*: BOOL;
	bSafeCommErr AT %I*: BOOL;
	bSafeRedLedOutput AT %Q*:BOOL; // safety output signal for EL2809 
	bSafeRedLedInput AT %I*:BOOL; // safety red led reception signal for ouput signal imported from EL6910
	bSafeRestartSignal AT %Q*: BOOL; //restart signal for safeESTop FB
	bSafeRestartSignalInput AT %I*: BOOL; //restart signal*)
END_VAR

// ---- GVLs/IO.TcGVL
{attribute 'qualified_only'}
VAR_GLOBAL
	
	bRun AT %I* 	: BOOL;
	bRestart AT %I* : BOOL;
	
END_VAR

// ---- POUs/FB_ClockPulse.TcPOU
FUNCTION_BLOCK FB_ClockPulse
VAR_INPUT
	bStart:BOOL;
	delOn: TIME:=T#500MS;
	delOff: TIME:= T#200MS;
END_VAR
VAR_OUTPUT
	bExecuteClock: BOOL;
END_VAR
VAR
	fbTimer1, fbTimer2: TON;
END_VAR

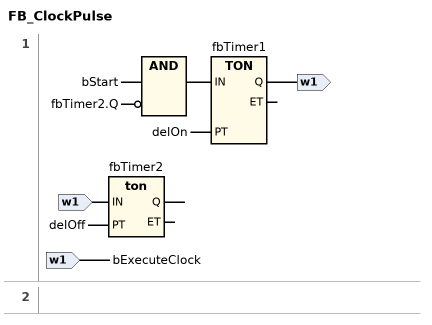
// NETWORK 1
fbTimer1(IN := bStart AND NOT fbTimer2.Q, PT := delOn); // TON
fbTimer2(IN := fbTimer1.Q, PT := delOff); // ton
bExecuteClock := fbTimer1.Q;

// NETWORK 2

END_FUNCTION_BLOCK

// ---- POUs/MAIN.TcPOU
PROGRAM MAIN
VAR
END_VAR


// Enable LED for VISION
IF GVL.bLedEnableVirtualInputButton THEN
	GVL.bLedEnableEL2xxx := TRUE;
ELSE
	GVL.bLedEnableEL2xxx:= FALSE;
END_IF

PRG_Thermocouple();
PRG_PowerMeasurement();
PRG_MotorDrive();
PRG_VfdModbusRtu();
PRG_LoadcellScaling();
PRG_PLCModbusRTU();
PRG_PneumaticValves();
PRG_SafetyLightCurtain();

END_PROGRAM

// ---- POUs/PRG_Thermocouple.TcPOU
PROGRAM PRG_Thermocouple
VAR
	fTemp: REAL;
	nMode: INT;
	bOffStat: BOOL;
	fbTONSwMode: TON;
	fbRTrigSwOn: R_TRIG;
	fbRTrigSwOff: R_TRIG;
	bSwOnVirtual: BOOL;
	bSwOffVirtual: bool;
END_VAR

fTemp := GVL.nTemp/10;
fbRTrigSwOn(CLK:= GVL.bSwOn OR bSwOnVirtual, Q=> );
fbRTrigSwOff(CLK:= GVL.bSwOff OR bSwOffVirtual, Q=> );

CASE nMode OF
	0: //Manual mode
		IF NOT GVL.bLight THEN
			fbTONSwMode(IN:= TRUE, PT:= T#10S, Q=> , ET=> );
		END_IF
		
		IF fbTONSwMode.Q THEN
			fbTONSwMode(IN:= FALSE);
			nMode := 1;
		END_IF
		
	1: //Automatic mode
		IF fTemp <= 26 THEN
			GVL.bLight := TRUE;
			GVL.bFan := FALSE;
		END_IF
		
		IF fTemp > 28 THEN
			GVL.bLight := FALSE;
			GVL.bFan := TRUE;
		END_IF
		
		IF fbRTrigSwOn.Q OR fbRTrigSwOff.Q THEN
			GVL.bFan := FALSE;
			nMode := 0;
		END_IF
END_CASE

IF fbRTrigSwOn.Q THEN
	fbTONSwMode(IN:= FALSE);
	GVL.bLight := TRUE;
END_IF

IF fbRTrigSwOff.Q THEN
	GVL.bLight := FALSE;
END_IF

END_PROGRAM

// ---- POUs/PRG_PowerMeasurement.TcPOU
PROGRAM PRG_PowerMeasurement
VAR
	fActivePowerAbs: REAL;
	fIL1Abs: REAL;
END_VAR

fActivePowerAbs := ABS(GVL.fActivePower);
fIL1Abs := ABS(GVL.fIL1);

END_PROGRAM

// ---- POUs/PRG_MotorDrive.TcPOU
PROGRAM PRG_MotorDrive
VAR
	fbEnableAxes: FB_EnableAxes;
	fbHalt1: MC_Halt;
	fbMoveVelocityFw: MC_MoveVelocity;
	fbMoveVelocityBw: MC_MoveVelocity;
	fbTON1: TON;
	fbRTrigMoveFw: R_TRIG;
	fbRTrigMoveBw: R_TRIG;
	fbRTrigHalt: R_TRIG;
	nAutoState: INT;
	nSpeed: INT := 400; //degrees/sec
	bButtonFwVirtual: BOOL:=FALSE;
	bButtonHaltVirtual: BOOL:=FALSE;
	bEnableServo: BOOL;
END_VAR

fbEnableAxes.bEnableAxes := bEnableServo;
fbRTrigMoveFW(CLK:=GVL.bButtonFw OR bButtonFwVirtual, Q=>);
fbRTrigMoveBW(CLK:=GVL.bButtonBw, Q=>);
fbRTrigHalt(CLK:=GVL.bButtonHalt OR bButtonHaltVirtual, Q=>);

IF fbRTrigMoveFw.Q THEN
	fbHalt1.Execute := FALSE;
	fbMoveVelocityBw.Execute := FALSE;
	fbMoveVelocityFw.Execute := TRUE;
END_IF

IF fbRTrigMoveBw.Q THEN
	fbHalt1.Execute := FALSE;
	fbMoveVelocityFw.Execute := FALSE;
	fbMoveVelocityBw.Execute := TRUE;
END_IF

IF fbRTrigHalt.Q THEN
	fbHalt1.Execute := TRUE;
	fbMoveVelocityFw.Execute := FALSE;
	fbMoveVelocityBw.Execute := FALSE;
END_IF

IF GVL.bButtonAuto THEN
	CASE nAutoState OF
		0: //Initialize auto motion
			fbHalt1.Execute := FALSE;
			fbMoveVelocityFw.Execute := FALSE;
			fbMoveVelocityBw.Execute := FALSE;
			nAutoState := 1;
		1: //Move forward
			fbTON1(IN:=TRUE, PT:=T#4S, Q=>, ET=>);
			fbMoveVelocityFw.Execute := TRUE;
			IF fbTON1.Q THEN
				fbTON1(IN:=FALSE);
				nAutoState := 2;	
			END_IF
		2: //Halt
			fbTON1(IN:=TRUE, PT:=T#2S, Q=>, ET=>);
			fbMoveVelocityFw.Execute := FALSE;
			fbHalt1.Execute := TRUE;
			IF fbTON1.Q THEN
				fbTON1(IN:=FALSE);
				nAutoState := 3;	
			END_IF
		3: //Move backward
			fbTON1(IN:=TRUE, PT:=T#4S, Q=>, ET=>);
			fbHalt1.Execute := FALSE;
			fbMoveVelocityBw.Execute := TRUE;
			IF fbTON1.Q THEN
				fbTON1(IN:=FALSE);
				nAutoState := 4;	
			END_IF
		4: //Halt again
			fbTON1(IN:=TRUE, PT:=T#2S, Q=>, ET=>);
			fbMoveVelocityBw.Execute := FALSE;
			fbHalt1.Execute := TRUE;
			IF fbTON1.Q THEN
				fbTON1(IN:=FALSE);
				nAutoState := 0;	
			END_IF
	END_CASE
END_IF

A_EnableAxes();
A_MoveVelocityFw();
A_MoveVelocityBw();
A_Halt();

ACTION A_EnableAxes:
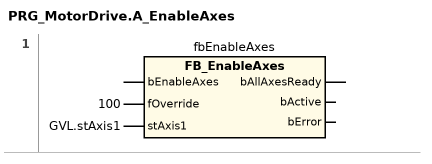
// NETWORK 1
fbEnableAxes(fOverride := 100, stAxis1 := GVL.stAxis1); // FB_EnableAxes
END_ACTION

ACTION A_Halt:
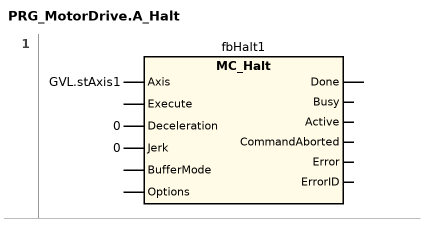
// NETWORK 1
fbHalt1(Axis := GVL.stAxis1, Deceleration := 0, Jerk := 0); // MC_Halt
END_ACTION

ACTION A_MoveVelocityBw:
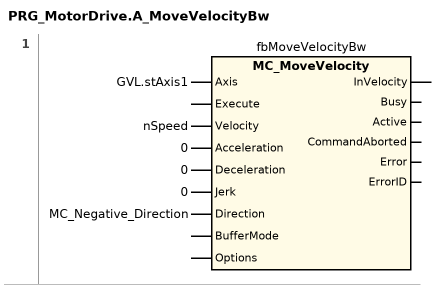
// NETWORK 1
fbMoveVelocityBw(
    Axis := GVL.stAxis1,
    Velocity := nSpeed,
    Acceleration := 0,
    Deceleration := 0,
    Jerk := 0,
    Direction := MC_Negative_Direction); // MC_MoveVelocity
END_ACTION

ACTION A_MoveVelocityFw:
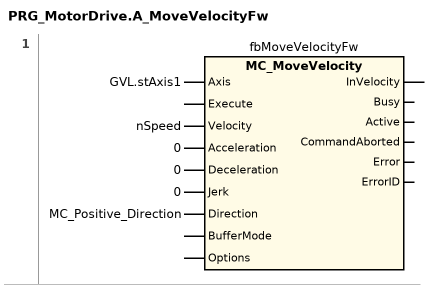
// NETWORK 1
fbMoveVelocityFw(
    Axis := GVL.stAxis1,
    Velocity := nSpeed,
    Acceleration := 0,
    Deceleration := 0,
    Jerk := 0,
    Direction := MC_Positive_Direction); // MC_MoveVelocity
END_ACTION

END_PROGRAM

// ---- POUs/PRG_VfdModbusRtu.TcPOU
PROGRAM PRG_VfdModbusRtu
VAR
	fbVfdMb: ModbusRtuMaster_KL6x22B;
	fbRTrigWrite: R_TRIG;
	fbRTrigEnable: R_TRIG;
	fbRTrigDisable: R_TRIG;
	fbRTrigReverseMotor: R_TRIG;
	fbRTrigSetFrequency: R_TRIG;
	fbTON: TON;
	fbTON1: TON;
	fbTON2: TON;
	fbTON3: TON;
	wQty: WORD := 1;
	wMbAddr: WORD;
	wCmd: WORD;
	wCmdPrev: WORD;
	bWrite: BOOL;
	bEnablePulse: BOOL;
	bPendingFlag: BOOL;
	bPulse: BOOL;
	bSetFreqCmd: BOOL;
	nSetFreqState: INT;
	nSetFreqVal: WORD;
END_VAR

fbRTrigWrite(CLK:=bWrite, Q=>);
fbRTrigEnable(CLK:= GVL.bRunVfd OR GVL.bEnable, Q=>);
fbRTrigDisable(CLK:= GVL.bStopVfd OR GVL.bDisable, Q=>);
fbRTrigReverseMotor(CLK:= GVL.bReverseMotor, Q=> );
fbRTrigSetFrequency(CLK:= GVL.bSetMotorFrequency, Q=> );

//Enable control word
IF fbRTrigEnable.Q THEN
	IF bWrite THEN
		bPendingFlag := TRUE; //Raise flag for pending command
	ELSE
		bWrite := TRUE;
	END_IF
	bEnablePulse := TRUE;
	wMbAddr := 417;
	wCmd := 32771;
END_IF

//Disable control word
IF fbRTrigDisable.Q THEN
	IF bWrite THEN
		bPendingFlag := TRUE; //Raise flag for pending command
	ELSE
		bWrite := TRUE;
	END_IF
	
	bEnablePulse := FALSE;
	wMbAddr := 417;
	wCmd := 0;
END_IF

//Reverse motor
IF fbRTrigReverseMotor.Q THEN
	IF bWrite THEN
		bPendingFlag := TRUE; //Raise flag for pending command
	ELSE
		bWrite := TRUE;
	END_IF
	bEnablePulse := TRUE;
	wMbAddr := 417;
	wCmd := 32777;	
END_IF

//Set motor frequency
IF fbRTrigSetFrequency.Q THEN
	bSetFreqCmd := TRUE;
	wCmdPrev := wCmd;
END_IF

IF bSetFreqCmd THEN
	CASE nSetFreqState OF
		0: //Set frequency
			IF bWrite THEN
				bPendingFlag := TRUE; //Raise flag for pending command
			ELSE
				bWrite := TRUE;
			END_IF
			bEnablePulse := FALSE;
			wMbAddr := 215;
			wCmd := nSetFreqVal*10;
			IF fbVfdMb.BUSY THEN
				nSetFreqState := 1;
			END_IF
		1: //Continue the previous command
			bSetFreqCmd := FALSE;
			IF wCmdPrev <> 0 THEN
				bEnablePulse := TRUE; //Short delay before pulse starts
				wMbAddr := 417;
				wCmd := wCmdPrev;
			END_IF
			nSetFreqState := 0;
	END_CASE
END_IF
//Keep sending enable signal to avoid watchdog error
fbTON1(IN:= bEnablePulse AND NOT fbTON2.Q, PT:= T#600MS, Q=> bPulse, ET=> ); //Pulse off time
fbTON2(IN:= fbTON1.Q, PT:= T#300MS, Q=> , ET=> );//Pulse on time

CASE wCmd OF
	32771: //Run motor forward
		GVL.bEnable := bPulse;
	32777: //Reverse motor
		GVL.bReverseMotor := bPulse;
END_CASE

IF bWrite THEN
	fbTON(IN:= bWrite, PT:= T#100MS, Q=> , ET=> );
END_IF

//Reset bWrite after a short delay
IF fbTON.Q THEN
	fbTON(IN:=FALSE);
	bWrite := FALSE;
END_IF

//Handle the raised pending flag
IF bPendingFlag AND NOT bWrite THEN
	fbTON3(IN:= TRUE, PT:= T#100MS, Q=> , ET=> );
END_IF

IF fbTON3.Q THEN
	fbTON3(IN:= FALSE);
	bPendingFlag := FALSE;
	bWrite := TRUE;
END_IF

fbVfdMb.WriteRegs(
	UnitID:= 1, 
	Quantity:= wQty, 
	MBAddr:= wMbAddr, 
	cbLength:= SIZEOF(wCmd), 
	pMemoryAddr:= ADR(wCmd), 
	Execute:= bWrite,//fbRTrigWrite.Q, 
	Timeout:= T#1S, 
	BUSY=> , 
	Error=> , 
	ErrorId=> , 
	cbRead=> );

END_PROGRAM

// ---- POUs/PRG_LoadcellScaling.TcPOU
PROGRAM PRG_LoadcellScaling
VAR
	bActivateLoadcellScaling AT %I*: BOOL;
	bDeactivateLoadcellScaling AT %I*:BOOL;
	bActiveState: BOOL;
	bZeroing: BOOL;
	bSet300Gr: BOOL;
	nMinValue: DINT:=430;
	nMaxValue: DINT:=1100;
END_VAR

// Detect /deactivate state for function 
IF 	bActivateLoadcellScaling AND NOT bDeactivateLoadcellScaling THEN
	bActiveState:=TRUE;
ELSIF 	bDeactivateLoadcellScaling AND NOT bActivateLoadcellScaling THEN
	bActiveState:=FALSE;
END_IF

// Funtion execute
IF bActiveState THEN
	IF bZeroing THEN
		nMinValue:= GVL.uLoadCellRawValue;
	END_IF
	IF bSet300Gr THEN
		nMaxValue:= GVL.uLoadCellRawValue;
	END_IF
	GVL.uLoadCellScaledValue := F_Scale(GVL.uLoadCellRawValue, 0.0, 0.3, nMinValue, nMaxValue);
ELSE
	GVL.uLoadCellScaledValue:= 0.0;
END_IF

END_PROGRAM

// ---- POUs/PRG_PLCModbusRTU.TcPOU
PROGRAM PRG_PLCModbusRTU
VAR
	bActivatePlcModbusWriteReg AT %I*: BOOL;
	bDeactivatePlcModbusWriteReg AT %I*: BOOL;
	bActiveState : BOOL;
	
	fbStrAscConversion: FB_StrASCConversion;
	fbModbusMaster: ModbusRtuMasterV2_KL6x22B;
	sWriteErrorId: MODBUS_ERRORS;
	bBusyState: BOOL := FALSE;
	
	fbRTrigClockPulse: R_TRIG;
	fbRTrigExecuteFirstReg: R_TRIG;
	fbRTrigExecuteSingleReg: R_TRIG;
	fbClockPulse: FB_ClockPulse;
	fbUpdateCycleClockPulse: FB_ClockPulse;
	nCount : INT;  // Send particular register decision
	nCountPulse : INT;
	// Modbus properties
	mB_unitId: BYTE:= 10;
	mB_unitIdForHmi: BYTE:= 8;
	mB_quantity_coils: WORD:=2;
	mB_quantity_regs: WORD:=10;
	mB_quantity_regForHmi: WORD:=1;
	mB_addr_bits: WORD:=00;
	
	mB_addr_1st10regs: WORD:=40;
	mB_addr_2nd10regs: WORD:=50;
	mB_addr_singleRegForHmi: WORD:=0;

	
	// Holding register declaration
	aWriteValueRegs0: ARRAY[0..19] OF WORD;
	aValue1st10Regs: ARRAY[0..9] OF WORD;
	aValue2nd10Regs: ARRAY[0..9] OF WORD;
	i : INT;
	bWrite: BOOL:=FALSE;
	bTurnOnPulse:BOOL:=FALSE;
	// Compressed form of coil registers
	wWriteValueBits: WORD; //BIT0|BIT1|XXXXXXXXX	

	bPlaceHolder: BOOL;
	wValueSingleRegForHmi: WORD:= 1;
	nChangeLangueCycle: INT:= 30;
	tLanguageCycle: TIME:= T#30S;
	bModeAuto: BOOL:=TRUE;
	bExecuteSingleReg: BOOL;
END_VAR

// Change INTEGER to TIME
IF nChangeLangueCycle = 0 THEN
	nChangeLangueCycle:= 1;
END_IF
tLanguageCycle:= INT_TO_TIME(nChangeLangueCycle*1000);

// Divide the array into two arrays
FOR i := 0 TO 19 DO
    IF i <= 9 THEN
        aValue1st10Regs[i] := aWriteValueRegs0[i];
    ELSE
        aValue2nd10Regs[i - 10] := aWriteValueRegs0[i];
    END_IF;
END_FOR;
// update cycle clock pulse creation
fbUpdateCycleClockPulse(bStart:= TRUE, delOn:= tLanguageCycle, delOff:= T#200MS, bExecuteClock => );
fbRTrigExecuteSingleReg(CLK:= fbUpdateCycleClockPulse.bExecuteClock, Q =>);
// Convert STRING to ARRAY OF BYTE in ASCII TYPE
fbStrAscConversion(sText:=GVL.sInputFromHMI,aASCIIRes => aWriteValueRegs0);

// Detect /deactivate state for function 
IF 	bActivatePlcModbusWriteReg AND NOT bDeactivatePlcModbusWriteReg THEN
	bActiveState:=TRUE;
ELSIF 	bDeactivatePlcModbusWriteReg AND NOT bActivatePlcModbusWriteReg THEN
	bActiveState:=FALSE;
END_IF

IF bActiveState THEN
	fbModbusMaster.WriteSingleRegister(
		UnitID:= mB_unitIdForHmi,
		Quantity:= mB_quantity_regForHmi, 
		MBAddr:= mB_addr_singleRegForHmi, 
		cbLength:= SIZEOF(wValueSingleRegForHmi),
		pMemoryAddr:= ADR(wValueSingleRegForHmi),
		Execute:= bExecuteSingleReg, 
		Timeout:= T#1500MS, 
		BUSY=> bBusyState, 
		Error=> , 
		ErrorId=> sWriteErrorId, 
		cbRead=>
	);
	bPlaceHolder:=TRUE;	
END_IF

IF bModeAuto THEN
	bExecuteSingleReg:= fbUpdateCycleClockPulse.bExecuteClock;
ELSE
	bExecuteSingleReg:= GVL.bExecuteWriteSingleRegForHmi;
END_IF

IF fbRTrigExecuteSingleReg.Q THEN
	IF wValueSingleRegForHmi <= 2 THEN
		wValueSingleRegForHmi:= wValueSingleRegForHmi+1;
	ELSE
			wValueSingleRegForHmi:= 1;	
	END_IF
END_IF

A_WriteCoils();

ACTION A_WriteCoils:
// ------Write coils-------
// Convert Bit 0 and Bit 1 to WORD
IF GVL.bModbusCoilBit0 THEN
	IF GVL.bModbusCoilBit1 THEN
		wWriteValueBits := 3;
	ELSE
		wWriteValueBits := 1;
	END_IF
ELSE
	IF GVL.bModbusCoilBit1 THEN
		wWriteValueBits := 2;
	ELSE
		wWriteValueBits := 0;
	END_IF
END_IF


fbModbusMaster.WriteMultipleCoils(
	UnitID:= mB_unitId, 
	Quantity:= mB_quantity_coils, 
	MBAddr:= mB_addr_bits, 
	cbLength:= SIZEOF(wWriteValueBits), 
	pMemoryAddr:= ADR(wWriteValueBits), 
	Execute:= GVL.bExecuteWriteCoils, 
	Timeout:= T#1000MS, 
	BUSY=> bBusyState, 
	Error=> , 
	ErrorId=> sWriteErrorId, 
	cbRead=>
);
END_ACTION

ACTION A_WriteRegHmi:

END_ACTION

ACTION A_WriteRegs:
//-----Write registers-------
//==> Divide into 2 arrays[0..9] due to unstable sending sequences when try to push 20 registers subsequently

	// Trigger for SEND button and clock pulse
fbRTrigExecuteFirstReg(CLK:= GVL.bExecuteWriteRegs0, Q =>);
fbRTrigClockPulse(CLK:= fbClockPulse.bExecuteClock, Q=>);

IF fbRTrigExecuteFirstReg.Q THEN
		bWrite := TRUE;
END_IF

IF bWrite THEN
	bTurnOnPulse:=TRUE;
END_IF

// Activate clockpulse
fbClockPulse(bStart:= bTurnOnPulse,delON:= T#1600MS, bExecuteClock => );

IF nCount = 0  AND bWrite = TRUE THEN
//Write first 10 regs
	fbModbusMaster.WriteRegs(
		UnitID:= mB_unitId,
		Quantity:= mB_quantity_regs, 
		MBAddr:= mB_addr_1st10regs, 
		cbLength:= SIZEOF(aValue1st10Regs), 
		pMemoryAddr:= ADR(aValue1st10Regs), 
		Execute:= fbClockPulse.bExecuteClock, 
		Timeout:= T#1500MS, 
		BUSY=> bBusyState, 
		Error=> , 
		ErrorId=> sWriteErrorId, 
		cbRead=>
	);
	IF nCountPulse >= 1 THEN
		nCount:=1;
	ELSE
		IF fbRTrigClockPulse.Q THEN
			nCountPulse:= nCountPulse+1;
		END_IF
	END_IF
ELSIF nCount = 1 AND bWrite = TRUE THEN
// Write second 10 regs
	fbModbusMaster.WriteRegs(
		UnitID:= mB_unitId,
		Quantity:= mB_quantity_regs, 
		MBAddr:= mB_addr_2nd10regs, 
		cbLength:= SIZEOF(aValue2nd10Regs), 
		pMemoryAddr:= ADR(aValue2nd10Regs), 
		Execute:= fbClockPulse.bExecuteClock, 
		Timeout:= T#1500MS, 
		BUSY=> bBusyState, 
		Error=> , 
		ErrorId=> sWriteErrorId, 
		cbRead=>
	);
	IF nCountPulse = 2 THEN
		bTurnOnPulse:=FALSE;
	ELSIF nCountPulse >=3 AND bBusyState =FALSE THEN // Wait until FB fishishes its functiong, avoid being suspended at busy state
		nCount:=0;
		nCountPulse:=0;
		bWrite:=FALSE;
		bTurnOnPulse:=FALSE;
	END_IF
	
	IF fbRTrigClockPulse.Q THEN
		nCountPulse:= nCountPulse+1;
	END_IF
END_IF
END_ACTION

METHOD M_BoolWordConversion : WORD
VAR_INPUT
END_VAR
END_METHOD

END_PROGRAM

// ---- POUs/PRG_PneumaticValves.TcPOU
PROGRAM PRG_PneumaticValves
VAR
	bActivatePneumaticValves AT %I*: BOOL;
	bDeactivatePneumaticValves AT %I*:BOOL;
	bActiveState: BOOL;
END_VAR

// Detect activate/deactivate state for function 
IF 	bActivatePneumaticValves AND NOT bDeactivatePneumaticValves THEN
	bActiveState:=TRUE;
ELSIF
	bDeactivatePneumaticValves AND NOT bActivatePneumaticValves THEN
	bActiveState:=FALSE;
END_IF


// Function execution
IF bActiveState THEN
	// Valve 1
	IF GVL.bVirtualToggleButton1 THEN
		GVL.bValve1:=TRUE;
	ELSE
		GVL.bValve1:=FALSE;
	END_IF
	
	// Valve2
	IF GVL.bVirtualToggleButton2 THEN
		GVL.bValve2:=TRUE;
	ELSE
		GVL.bValve2:=FALSE;
	END_IF
	
	// Valve 3
	IF GVL.bVirtualToggleButton3 THEN
		GVL.bValve3:=TRUE;
	ELSE
		GVL.bValve3:=FALSE;
	END_IF
	
	
	// Valve 4
	IF GVL.bVirtualToggleButton4 THEN
		GVL.bValve4:=TRUE;
	ELSE
		GVL.bValve4:=FALSE;
	END_IF
	
	// Valve 5
	IF GVL.bVirtualToggleButton5 THEN
		GVL.bValve5:=TRUE;
	ELSE
		GVL.bValve5:=FALSE;
	END_IF
	
	// Valve 6
	IF GVL.bVirtualToggleButton6 THEN
		GVL.bValve6:=TRUE;
	ELSE
		GVL.bValve6:=FALSE;
	END_IF
END_IF

END_PROGRAM

// ---- POUs/PRG_SafetyLightCurtain.TcPOU
PROGRAM PRG_SafetyLightCurtain
VAR
	ErrAck AT %Q* 	: BOOL;
	RstEstop AT %Q* : BOOL;
	RunStop AT %Q* 	: BOOL;
	ComErr AT %I* 	: BOOL;
	FbErr AT %I* 	: BOOL;
	OutErr AT %I* 	: BOOL;
	
	a : R_TRIG;
	ncounter:INT:=0;
	
	//=== TwinSAFE Diagnostic ===//
	// target system
		wProjectCrc 	AT %I*	: WORD;
		idiSerialnumber AT %I* 	: UDINT;
	//Group 1
		fbTsGroup_1			: FB_TwinSafeGroupExt;
		stTsGroupInfo		: ST_TsGroupInfo;
	//TwinSAFE Connection
		fbTsConnection_EL6910	: FB_TwinSafeConnectionEL6910;
		fbTsConnection_EL1904	: FB_TwinSafeConnectionEL1904;
		fbTsConnection_EL2912	: FB_TwinSafeConnectionEL2912;
	//Twinsafe function block
		fbTsFB_Estop1			: FB_TwinSafeFB;
END_VAR

RstEstop:=IO.bRestart;
a(CLK:=IO.bRun , Q=> );
IF a.Q THEN
	ncounter:=ncounter+1;
	IF ncounter >1 THEN
		ncounter:=0;
	END_IF
END_IF

IF ncounter = 1 THEN
	RunStop:=TRUE;
	ELSE RunStop:=FALSE;
END_IF

//Diagnostic
//TwinSAFE (Group 1)
fbTsGroup_1(
	bRun:= IO.bRun, 
	bErrAck:= ErrAck, 
	sName:= 'Gr01_Estop');
//TwinSAFE connection
fbTsConnection_EL6910(tCoEReadCycle :=T#2S);
fbTsConnection_EL1904(tCoEReadCycle	:=T#2S) ;
fbTsConnection_EL2912(tCoEReadCycle	:=T#2S);
//Twinsafe Function Block
fbTsFB_Estop1(
	sName:= 'FBEstop1', 
	eFBType:= E_TsFbType.FB_TYPE_ESTOP, 
	nFbId:= 1);

END_PROGRAM

// ---- POUs/TwinSAFE/FB_TwinSafeConnectionEL2912.TcPOU
FUNCTION_BLOCK FB_TwinSafeConnectionEL2912
(*******************************************************************************************************
Description			:	Evaluate a TwinSAFE connection status and diagnosis to an EtherCAT terminal
Supported terminals : 	EL2912
Documentation 		:	EL2912 TwinSAFE potential supply terminal with 4 fail-safe inputs and 1 fail-safe output
Version/Date 		:	V1.1.0/20.12.2021
Required libraries 	: 	TcSystem.lib (Tc2_System), TcEtherCAT.lib (Tc2_EtherCAT)
********************************************************************************************************)
VAR_INPUT
	
	tCoEReadCycle							:TIME 	:= T#0MS;				(* Read cycle CoE-Data, e.g. temperature *)
	bLogicTerminal							:BOOL;
	
END_VAR
VAR_OUTPUT

	stInfoData						AT %I*	:ST_TsConnectionInfoEL2912;		(* [TwinSAFE logic] e.g. EL69xx \ Connection Info Data \ [Path] Info Data*)
	nEcSlaveState					AT %I*	:UINT ;							(* EL2911 \ InfoData \ State *)
	stEcAdsAddr						AT %I*	:ST_AdsAddr;					(* EL2911 \ InfoData \ AdsAddr *)
	
	stTsSlaveInfo							:ST_TsSlaveInfoEL2912;

END_VAR
VAR

(* act_ConnectionDiag *)
	nDiag0_3								:BYTE;

(* act_ReadDiagObjects *)
	eReadDiagObjState						:E_TsCycleDiagObj;
	eReadDiagObjErrStep						:E_TsCycleDiagObj := E_TsCycleDiagObj.eCycleDiagObj_NoError;
	bReadDiagObjError						:BOOL;							(* Error in the diagnosis objects read cycle *)  
	bReadDiagObjReset						:BOOL;							(* Reset the diagnosis objects read cycle error *)
	fbTimer									:TON;
	fbEcCoeSdoRead							:FB_EcCoESdoReadEx;
	stDiagObjects							:ST_TsDiagObjectsEL2912;

(* act_EcSlaveIdentify *)
	fbEcGetSlaveName						:FB_EcGetSlaveName;

END_VAR
VAR CONSTANT
	
(* act_ReadDiagObjects *)
	nWarningLevelTemp1						:INT	:= 85;					(* Temperature 1 warning level [°C] *)
	nWarningLevelTemp2						:INT	:= 85;					(* Temperature 2 warning level [°C] *)

END_VAR
(* End *)

(* Function Block TwinSAFE connection status and diagnosis for EP1957 Terminals *)

(* THIS CODE IS ONLY AN EXAMPLE - YOU HAVE TO CHECK APTITUDE FOR YOUR APPLICATION *)

	(* Identify the EtherCAT slave *)
		act_EcSlaveIdentify();

	(* Evaluate the connection state *)
		act_ConnectionState();
	
	(* Evaluate the connection diagnosis *)
		act_ConnectionDiag();
	
	(* Evaluate the signals *)
		act_Signals();
	
	(* Evaluate the Terminal temperatures and diagnostic objects *)
	IF stTsSlaveInfo.bSlaveIdentify
		THEN
			act_ReadDiagObjects();
		ELSE
			eReadDiagObjState := E_TsCycleDiagObj.eCycleDiagObj_Init;
		END_IF
	
(* End *)

ACTION act_ConnectionDiag:
(* Evaluate the connection diagnosis *)

	(* Evaluate Bit 0..3 *)
	nDiag0_3 := USINT_TO_BYTE(stInfoData.nDiag) AND 16#0F;

	CASE nDiag0_3 OF
		0:		stTsSlaveInfo.sDiag := 'No error';
		1:		stTsSlaveInfo.sDiag := 'Invalid command';
		2:		stTsSlaveInfo.sDiag := 'Unknown command';
		3:		stTsSlaveInfo.sDiag := 'Invalid connection ID';
		4:		stTsSlaveInfo.sDiag := 'Invalid CRC';
		5:		stTsSlaveInfo.sDiag := 'Watchdog time elapsed';
		6:		stTsSlaveInfo.sDiag := 'Invalid FSOE address';
		7:		stTsSlaveInfo.sDiag := 'Invalid data';
		8:		stTsSlaveInfo.sDiag := 'Invalid communication parameter length';
		9:		stTsSlaveInfo.sDiag := 'Invalid communication parameters';
		10:		stTsSlaveInfo.sDiag := 'Invalid user parameter length';
		11:		stTsSlaveInfo.sDiag := 'Invalid user parameter';
		12:		stTsSlaveInfo.sDiag := 'FSoE master reset';
		13:		stTsSlaveInfo.sDiag := 'Module err detected on slave, with option "Module error is ComError" activated';
		14:		stTsSlaveInfo.sDiag := 'Module err detected on EL290x, with option "Error acknowledge active" activated';
		15:		stTsSlaveInfo.sDiag := 'Slave not yet started, or unexpected error argument';
	END_CASE

	(* Evaluate Bit 4..7 *)
	stTsSlaveInfo.sFault:='';

	IF stInfoData.nDiag.4 
	THEN
		stTsSlaveInfo.sFault	:= 'FSoE slave error detected - '; 
	END_IF

	IF stInfoData.nDiag.5 
	THEN
		stTsSlaveInfo.sFault	:= concat(stTsSlaveInfo.sFault,'FSoE slave reports Failsafe Value active - ');
	END_IF

	IF stInfoData.nDiag.6 
	THEN
		stTsSlaveInfo.sFault	:= concat(stTsSlaveInfo.sFault,'StartUp - ');
	END_IF

	IF stInfoData.nDiag.7 
	THEN
		stTsSlaveInfo.sFault	:= concat(stTsSlaveInfo.sFault, 'FSoE master reports Failsafe Value active');
	END_IF
		
	(* Error *)
	stTsSlaveInfo.bError := stInfoData.nDiag <> 0;

(* End *)
END_ACTION

ACTION act_ConnectionState:
(* Evaluate the connection state *)

	CASE stInfoData.nState OF
		100:	stTsSlaveInfo.sState := 'Reset state';
		101:	stTsSlaveInfo.sState := 'Session state';
		102:	stTsSlaveInfo.sState := 'Connection state';
		103:	stTsSlaveInfo.sState := 'Parameter state';
		104:	stTsSlaveInfo.sState := 'Data state';
		105:	stTsSlaveInfo.sState := 'Shutdown state';
		106:	stTsSlaveInfo.sState := 'Shutdown state deactive';
	ELSE
		IF bLogicTerminal
		THEN
			stTsSlaveInfo.sState := 'Master';
		ELSE
			stTsSlaveInfo.sState := 'unknown';
		END_IF
	END_CASE
	
(* End *)
END_ACTION

ACTION act_DiagObjectsBits:
(* act_TsDiagObjectsBits *)
(*
	stTsDiagObjectsBitsEL1904.bErrInput1		 			 := stDiagObjects.nSensorTestError.0;
	stTsDiagObjectsBitsEL1904.bErrInput2		 			 := stDiagObjects.nSensorTestError.1;
	stTsDiagObjectsBitsEL1904.bErrInput3		 			 := stDiagObjects.nSensorTestError.2;
	stTsDiagObjectsBitsEL1904.bErrInput4		 			 := stDiagObjects.nSensorTestError.1;
	
	stTsDiagObjectsBitsEL1904.bErrFirstInputPair 			 := stDiagObjects.nDuringTwoChannelEvaluationError.0;
	stTsDiagObjectsBitsEL1904.bErrSecondInputPair 			 := stDiagObjects.nDuringTwoChannelEvaluationError.1;

	stTsDiagObjectsBitsEL1904.bMatOpModeErrFirstInputPair	 := stDiagObjects.nMatModeInputPairDisagreeError.0 
																	AND stDiagObjects.nMatModeInputPairDisagreeError.1;
	stTsDiagObjectsBitsEL1904.bMatOpModeErrSecondInputPair	 := stDiagObjects.nMatModeInputPairDisagreeError.2 
																	AND stDiagObjects.nMatModeInputPairDisagreeError.3;

	stTsDiagObjectsBitsEL1904.bMatOpModeExtSupplyErrInput1 	 := stDiagObjects.nMatModeExternalSupplyError.0;
	stTsDiagObjectsBitsEL1904.bMatOpModeExtSupplyErrInput2 	 := stDiagObjects.nMatModeExternalSupplyError.1;
	stTsDiagObjectsBitsEL1904.bMatOpModeExtSupplyErrInput3 	 := stDiagObjects.nMatModeExternalSupplyError.2;
	stTsDiagObjectsBitsEL1904.bMatOpModeExtSupplyErrInput4 	 := stDiagObjects.nMatModeExternalSupplyError.3;
*)
(* End *)
END_ACTION

ACTION act_EcSlaveIdentify:
(* Identify the EtherCAT slave *)

	IF NOT nEcSlaveState.3
	THEN
		stTsSlaveInfo.bSlaveIdentify  := FALSE;
		stTsSlaveInfo.bSlaveTypeError := FALSE;
		stTsSlaveInfo.sEcSlaveType    := '';
	END_IF

	IF nEcSlaveState.3
		AND NOT stTsSlaveInfo.bSlaveIdentify
		AND NOT stTsSlaveInfo.bSlaveTypeError
 		AND F_CreateAmsNetId(stEcAdsAddr.netId) <> '0.0.0.0.0.0' 
		AND stEcAdsAddr.port <> 0
	THEN

		fbEcCoeSdoRead(
			sNetId			:= 	F_CreateAmsNetId(stEcAdsAddr.netId),
			nSlaveAddr		:= 	stEcAdsAddr.port,
			nSubIndex		:= 	0,
			nIndex			:= 	16#1008,
			pDstBuf			:= 	ADR(stTsSlaveInfo.sEcSlaveType),
			cbBufLen		:= 	SIZEOF(stTsSlaveInfo.sEcSlaveType),
			bExecute		:= 	TRUE,
			tTimeout		:= 	DEFAULT_ADS_TIMEOUT);
	

		fbEcGetSlaveName(
			bExecute		:=	TRUE, 
			sNetId			:=	F_CreateAmsNetId(stEcAdsAddr.netId), 
			nSlaveAddr		:=	stEcAdsAddr.port, 
			tTimeout		:=	DEFAULT_ADS_TIMEOUT, 
			bBusy			=>	, 
			sSlaveName		=>	stTsSlaveInfo.sEcSlaveName, 
			bError			=>	, 
			nErrId			=>	);

		IF NOT fbEcCoeSdoRead.bBusy
			AND NOT fbEcCoeSdoRead.bError
			AND NOT fbEcGetSlaveName.bBusy
			AND NOT fbEcGetSlaveName.bError
		THEN
		
			fbEcCoeSdoRead(bExecute := FALSE); 
			fbEcGetSlaveName(bExecute := FALSE); 

			IF stTsSlaveInfo.sEcSlaveType = 'EL2912' 
				AND fbEcGetSlaveName.sSlaveName <> ''
			THEN
				stTsSlaveInfo.bSlaveIdentify := TRUE;
			ELSE
				stTsSlaveInfo.bSlaveTypeError := TRUE;
			END_IF

		ELSIF NOT fbEcCoeSdoRead.bBusy
			AND fbEcCoeSdoRead.bError
		OR (NOT fbEcGetSlaveName.bBusy
			AND fbEcGetSlaveName.bError)
		THEN
		
			fbEcCoeSdoRead(bExecute := FALSE); 
			fbEcGetSlaveName(bExecute := FALSE); 

		END_IF

	END_IF


	IF nEcSlaveState.3
		AND stTsSlaveInfo.bSlaveIdentify
			AND NOT stTsSlaveInfo.bSlaveAddressOk
	THEN
		// Read slave FSoE Address  (F980:01)
		// Read slave serial number (F980:02)
		// Read slave project CRC 	(F980:03)

			fbEcCoeSdoRead(
				sNetId			:= 	F_CreateAmsNetId(stEcAdsAddr.netId),
				nSlaveAddr		:= 	stEcAdsAddr.port,
				nSubIndex		:= 	1,
				nIndex			:= 	16#F980,
				pDstBuf			:= 	ADR(stTsSlaveInfo.stTsSlaveAddress),
				cbBufLen		:= 	SIZEOF(stTsSlaveInfo.stTsSlaveAddress),
				bExecute		:= 	TRUE,
				tTimeout		:= 	DEFAULT_ADS_TIMEOUT,
				bCompleteAccess	:= 	TRUE);

			IF NOT fbEcCoeSdoRead.bBusy 
				AND NOT fbEcCoeSdoRead.bError 
			THEN
				fbEcCoeSdoRead(bExecute := FALSE);
				stTsSlaveInfo.nEcSlaveFSoEAddr 		:= stTsSlaveInfo.stTsSlaveAddress.nEcSlaveFSoEAddr;
				stTsSlaveInfo.nEcSlaveSerialNumber 	:= TO_UDINT(stTsSlaveInfo.stTsSlaveAddress.nEcSlaveSerialNumber[0] OR SHL(TO_DWORD(stTsSlaveInfo.stTsSlaveAddress.nEcSlaveSerialNumber[1]),16));
				stTsSlaveInfo.nEcProjectCrc			:= stTsSlaveInfo.stTsSlaveAddress.nEcSlaveProjectCRC;
				stTsSlaveInfo.bSlaveAddressOk 		:= TRUE;
			ELSIF NOT fbEcCoeSdoRead.bBusy 
				AND fbEcCoeSdoRead.bError 
			THEN
				fbEcCoeSdoRead(bExecute := FALSE);
				stTsSlaveInfo.nEcSlaveFSoEAddr 		:= 0;
				stTsSlaveInfo.nEcSlaveSerialNumber 	:= 0;
			END_IF	
	
	END_IF
	
(* End *)
END_ACTION

ACTION act_ReadDiagObjects:
(* Evaluate the Terminal temperatures and diagnostic objects *)

	CASE eReadDiagObjState OF

		eCycleDiagObj_Init				:	(* Init *)	

